// TwinCAT 3 PLC project BAUK_EK_BMS_PLC
// ProgramVersion: 3.1.4024.0
// libraries:
//   Recipe Management, * (System)
//   Tc2_BABasic, * (Beckhoff Automation GmbH)
//   Tc2_DALI, * (Beckhoff Automation GmbH)
//   Tc2_Database, * (Beckhoff Automation GmbH)
//   Tc2_DMX, * (Beckhoff Automation GmbH)
//   Tc2_EnOcean, * (Beckhoff Automation GmbH)
//   Tc2_EtherCAT, * (Beckhoff Automation GmbH)
//   Tc2_SerialCom, * (Beckhoff Automation GmbH)
//   Tc2_Standard, * (Beckhoff Automation GmbH)
//   Tc2_System, * (Beckhoff Automation GmbH)
//   Tc2_Utilities, * (Beckhoff Automation GmbH)
//   Tc3_DALI, * (Beckhoff Automation GmbH)
//   Tc3_IotBase, * (Beckhoff Automation GmbH)
//   Tc3_JsonXml, * (Beckhoff Automation GmbH)
//   Tc3_MLL, * (Beckhoff Automation GmbH)
//   Tc3_Module, * (Beckhoff Automation GmbH)
// project tree:
//   BLINDS/ ADSReadCX9020.TcPOU, BackgroundComms.TcPOU, BlindControl.TcPOU (not stored), BlindStretch.TcPOU, ConvertBoolArrayToString.TcPOU, fConvertBoolArrayToString.TcPOU, PrgMqttCom_Blinds_Publisher.TcPOU, Selection.TcDUT (not stored), StructAdvancedBlindControl.TcDUT (not stored), StructBlindControl.TcDUT (not stored)
//   ENOCEAN/ EnOcean.TcPOU
//   / FastDmxUpdate.TcTTO, Global_Variables.TcGVL, MAIN.TcPOU, PlcTask.TcTTO (not stored)
//   HMI/ FileHandle.TcPOU, ReadCP67.TcPOU, ST_SignInTable.TcDUT (not stored), SwitchTable.TcDUT (not stored), TableTennisScoreCounter.TcPOU, TIMESTR_Strings.TcDUT, VariableHandleForHmi.TcPOU
//   LIGHTS/DALI/ Dali.TcPOU, LightControl.TcPOU, LightTable.TcDUT (not stored)
//   LIGHTS/DMX/ DMX.TcPOU, ST_RGB.TcDUT
//   ML/ CoffeePredictionML.TcPOU (not stored), FB_CoffeeFifo.TcPOU, MLtest.TcPOU (not stored)
//   POWER MONITORING/ CoffeType.TcDUT (not stored), FB_Latch.TcPOU (not stored), PrgMqttCom_PM_Subscriber.TcPOU, SQLDB.TcPOU (not stored), ST_EL3403_Data.TcDUT, ST_PHASE_DATA.TcDUT (not stored)
//   WIND TURBINE/ FB_SendWhatsappCallMeBot.TcPOU, FB_WeatherAPI_HTTP.TcPOU, FB_WatsAppResponse.TcPOU, FB_WindTurbineSim.TcPOU
//   WORKSHOP WALL/ PowerSupply.TcPOU, Pulse.TcPOU, ST_PsuDiagData.TcDUT, ST_PsuInfoData.TcDUT
// real-time tasks:
//   TASK PlcTask: cycle T#2ms, priority 20, ADS port 350
//   TASK FastDmxUpdate: cycle T#1ms, priority 1, ADS port 351
// I/O:
//   DEVICE CX2040 E-Bus, AmsNetId 192.168.56.1.2.1
//     CX2040 Supply [EK1200-5000 EtherCAT Power supply (2A E-Bus)]
//       Server Room EtherCAT Junction [EK1122 2 port EtherCAT junction]
//         Boardroom DMX Node [EK1100 EtherCAT Coupler (2A E-Bus)]
//           Cabinet LED Strip Control [EL6851 DMX Master]
//           Term 17 (EL9011) [EL9011 End Terminal]
//         24Vdc Power Supply On Test Wall [PS2001-2410-1001 Power supply (24V, 10A, 1-phase)]
//         OLD BLIND CONTROL [EK1100 EtherCAT Coupler (2A E-Bus)] (disabled)
//           Coffee Machine Power Monitor [EL3403 3Ch. Power Measuring]
//           Blind Control Staff Room [EL6001 Interface (RS232)]
//           Blind Control Communal Area [EL6001 Interface (RS232)]
//           Blind Control Boardroom [EL6001 Interface (RS232)]
//       E-Bus to K-Bus
// variable links:
//   BAUK_EK_BMS_PLC/BAUK_EK_BMS_PLC Instance <-> CX2040 E-Bus/CX2040 Supply/E-Bus to K-Bus
//     PlcTask Inputs/.stDALIInData/nData <-> Office DALI Light Control/Channel 1/Data In
//     PlcTask Inputs/.stDALIInData/nStatus <-> Office DALI Light Control/Channel 1/State
//     PlcTask Inputs/.stKL6581InData/CNODE <-> Office EnOcean Switch Control/Channel 1/Input CNODE
//     PlcTask Inputs/.stKL6581InData/DB{0..3} <-> Office EnOcean Switch Control/Channel 1/Input DB{0..3}  (4 links)
//     PlcTask Inputs/.stKL6581InData/ID{0..3} <-> Office EnOcean Switch Control/Channel 1/Input ID{0..3}  (4 links)
//     PlcTask Inputs/.stKL6581InData/ORG <-> Office EnOcean Switch Control/Channel 1/Input ORG
//     PlcTask Inputs/.stKL6581InData/STATUS <-> Office EnOcean Switch Control/Channel 1/Input STATUS
//     PlcTask Inputs/.stKL6581InData/nStatus <-> Office EnOcean Switch Control/Channel 1/Status
//     PlcTask Inputs/.stKL6811InData/nData <-> Office DALI Light Control/Channel 1/Data In
//     PlcTask Inputs/.stKL6811InData/nStatus <-> Office DALI Light Control/Channel 1/State
//     PlcTask Inputs/EnOcean.STEnOceanInData/nData <-> Office RS485 EnOcean Control/Channel 1/Data In 0
//     PlcTask Inputs/EnOcean.STEnOceanInData/nData @bit {8..80 step 8} <-> Office RS485 EnOcean Control/Channel 1/Data In {1..10}  (10 links)
//     PlcTask Inputs/EnOcean.STEnOceanInData/nStatus <-> Office RS485 EnOcean Control/Channel 1/Ser. State
//     PlcTask Outputs/.stDALIOutData/nCtrl <-> Office DALI Light Control/Channel 1/Ctrl
//     PlcTask Outputs/.stDALIOutData/nData <-> Office DALI Light Control/Channel 1/Data Out
//     PlcTask Outputs/.stKL6581OutData/CNODE <-> Office EnOcean Switch Control/Channel 1/Output CNODE
//     PlcTask Outputs/.stKL6581OutData/DB{0..3} <-> Office EnOcean Switch Control/Channel 1/Output DB{0..3}  (4 links)
//     PlcTask Outputs/.stKL6581OutData/ID{0..3} <-> Office EnOcean Switch Control/Channel 1/Output ID{0..3}  (4 links)
//     PlcTask Outputs/.stKL6581OutData/ORG <-> Office EnOcean Switch Control/Channel 1/Output ORG
//     PlcTask Outputs/.stKL6581OutData/STATUS <-> Office EnOcean Switch Control/Channel 1/Output STATUS
//     PlcTask Outputs/.stKL6581OutData/nControl <-> Office EnOcean Switch Control/Channel 1/Control
//     PlcTask Outputs/EnOcean.STEnOceanOutData/nCtrl <-> Office RS485 EnOcean Control/Channel 1/Ser. Ctrl
//     PlcTask Outputs/EnOcean.STEnOceanOutData/nData[{0..10}] <-> Office RS485 EnOcean Control/Channel 1/Data Out {0..10}  (11 links)
//   BAUK_EK_BMS_PLC/BAUK_EK_BMS_PLC Instance <-> CX2040 E-Bus/CX2040 Supply/Server Room EtherCAT Junction/24Vdc Power Supply On Test Wall
//     PlcTask Inputs/PowerSupply.amsAdr <-> InfoData/AdsAddr
//     PlcTask Inputs/PowerSupply.psuDcOk <-> PSU Inputs/DC OK
//     PlcTask Inputs/PowerSupply.psuError <-> PSU Inputs/Error
//     PlcTask Inputs/PowerSupply.psuInputUnderVoltage <-> PSU Inputs Device/Input undervoltage
//     PlcTask Inputs/PowerSupply.psuOutCurrent <-> PSU Inputs/Output current
//     PlcTask Inputs/PowerSupply.psuOutVoltage <-> PSU Inputs/Output voltage
//     PlcTask Inputs/PowerSupply.psuWarning <-> PSU Inputs/Warning
//     PlcTask Outputs/PowerSupply.psuDisableOutput <-> PSU Outputs/Disable output
//   BAUK_EK_BMS_PLC/BAUK_EK_BMS_PLC Instance <-> CX2040 E-Bus/CX2040 Supply/Server Room EtherCAT Junction/Boardroom DMX Node/Cabinet LED Strip Control
//     FastDmxUpdate Inputs/.stDMXInDataLinie01/bCyclicTxDDisabled <-> DMX Status/Cyclic TxD disabled
//     FastDmxUpdate Inputs/.stDMXInDataLinie01/bDefaultDataSent <-> DMX Status/Default data sent
//     FastDmxUpdate Inputs/.stDMXInDataLinie01/bFrameSentToggle <-> DMX Status/Frame sent toggle
//     FastDmxUpdate Inputs/.stDMXInDataLinie01/bReceiveToggle <-> DMX Status/Receive toggle
//     FastDmxUpdate Inputs/.stDMXInDataLinie01/bTransmitAccepted <-> DMX Status/Transmit accepted
//     FastDmxUpdate Inputs/.stDMXInDataLinie01/bTxPDOToggle <-> DMX Status/TxPDO Toggle
//     FastDmxUpdate Inputs/.stDMXInDataLinie01/byStartCode <-> DMX Status/Start code
//     FastDmxUpdate Inputs/.stDMXInDataLinie01/wChannelLength <-> DMX Status/Channel length
//     FastDmxUpdate Outputs/.stDMXOutDataLinie01/arrData <-> DMX Channel 1-64/Channel 1
//     FastDmxUpdate Outputs/.stDMXOutDataLinie01/arrData @bit 72 <-> DMX Channel 1-64/Channel 10
//     FastDmxUpdate Outputs/.stDMXOutDataLinie01/arrData @bit 80 <-> DMX Channel 1-64/Channel 11
//     FastDmxUpdate Outputs/.stDMXOutDataLinie01/arrData @bit 88 <-> DMX Channel 1-64/Channel 12
//     FastDmxUpdate Outputs/.stDMXOutDataLinie01/arrData @bit 96 <-> DMX Channel 1-64/Channel 13
//     FastDmxUpdate Outputs/.stDMXOutDataLinie01/arrData @bit 104 <-> DMX Channel 1-64/Channel 14
//     FastDmxUpdate Outputs/.stDMXOutDataLinie01/arrData @bit 112 <-> DMX Channel 1-64/Channel 15
//     FastDmxUpdate Outputs/.stDMXOutDataLinie01/arrData @bit 120 <-> DMX Channel 1-64/Channel 16
//     FastDmxUpdate Outputs/.stDMXOutDataLinie01/arrData @bit 128 <-> DMX Channel 1-64/Channel 17
//     FastDmxUpdate Outputs/.stDMXOutDataLinie01/arrData @bit 136 <-> DMX Channel 1-64/Channel 18
//     FastDmxUpdate Outputs/.stDMXOutDataLinie01/arrData @bit 144 <-> DMX Channel 1-64/Channel 19
//     FastDmxUpdate Outputs/.stDMXOutDataLinie01/arrData @bit 8 <-> DMX Channel 1-64/Channel 2
//     FastDmxUpdate Outputs/.stDMXOutDataLinie01/arrData @bit 152 <-> DMX Channel 1-64/Channel 20
//     FastDmxUpdate Outputs/.stDMXOutDataLinie01/arrData @bit 160 <-> DMX Channel 1-64/Channel 21
//     FastDmxUpdate Outputs/.stDMXOutDataLinie01/arrData @bit 168 <-> DMX Channel 1-64/Channel 22
//     FastDmxUpdate Outputs/.stDMXOutDataLinie01/arrData @bit 176 <-> DMX Channel 1-64/Channel 23
//     FastDmxUpdate Outputs/.stDMXOutDataLinie01/arrData @bit 184 <-> DMX Channel 1-64/Channel 24
//     FastDmxUpdate Outputs/.stDMXOutDataLinie01/arrData @bit 192 <-> DMX Channel 1-64/Channel 25
//     FastDmxUpdate Outputs/.stDMXOutDataLinie01/arrData @bit 200 <-> DMX Channel 1-64/Channel 26
//     FastDmxUpdate Outputs/.stDMXOutDataLinie01/arrData @bit 208 <-> DMX Channel 1-64/Channel 27
//     FastDmxUpdate Outputs/.stDMXOutDataLinie01/arrData @bit 216 <-> DMX Channel 1-64/Channel 28
//     FastDmxUpdate Outputs/.stDMXOutDataLinie01/arrData @bit 224 <-> DMX Channel 1-64/Channel 29
//     FastDmxUpdate Outputs/.stDMXOutDataLinie01/arrData @bit 16 <-> DMX Channel 1-64/Channel 3
//     FastDmxUpdate Outputs/.stDMXOutDataLinie01/arrData @bit 232 <-> DMX Channel 1-64/Channel 30
//     FastDmxUpdate Outputs/.stDMXOutDataLinie01/arrData @bit 240 <-> DMX Channel 1-64/Channel 31
//     FastDmxUpdate Outputs/.stDMXOutDataLinie01/arrData @bit 248 <-> DMX Channel 1-64/Channel 32
//     FastDmxUpdate Outputs/.stDMXOutDataLinie01/arrData @bit 256 <-> DMX Channel 1-64/Channel 33
//     FastDmxUpdate Outputs/.stDMXOutDataLinie01/arrData @bit 264 <-> DMX Channel 1-64/Channel 34
//     FastDmxUpdate Outputs/.stDMXOutDataLinie01/arrData @bit 272 <-> DMX Channel 1-64/Channel 35
//     FastDmxUpdate Outputs/.stDMXOutDataLinie01/arrData @bit 280 <-> DMX Channel 1-64/Channel 36
//     FastDmxUpdate Outputs/.stDMXOutDataLinie01/arrData @bit 288 <-> DMX Channel 1-64/Channel 37
//     FastDmxUpdate Outputs/.stDMXOutDataLinie01/arrData @bit 296 <-> DMX Channel 1-64/Channel 38
//     FastDmxUpdate Outputs/.stDMXOutDataLinie01/arrData @bit 304 <-> DMX Channel 1-64/Channel 39
//     FastDmxUpdate Outputs/.stDMXOutDataLinie01/arrData @bit 24 <-> DMX Channel 1-64/Channel 4
//     FastDmxUpdate Outputs/.stDMXOutDataLinie01/arrData @bit 312 <-> DMX Channel 1-64/Channel 40
//     FastDmxUpdate Outputs/.stDMXOutDataLinie01/arrData @bit 320 <-> DMX Channel 1-64/Channel 41
//     FastDmxUpdate Outputs/.stDMXOutDataLinie01/arrData @bit 328 <-> DMX Channel 1-64/Channel 42
//     FastDmxUpdate Outputs/.stDMXOutDataLinie01/arrData @bit 336 <-> DMX Channel 1-64/Channel 43
//     FastDmxUpdate Outputs/.stDMXOutDataLinie01/arrData @bit 344 <-> DMX Channel 1-64/Channel 44
//     FastDmxUpdate Outputs/.stDMXOutDataLinie01/arrData @bit 352 <-> DMX Channel 1-64/Channel 45
//     FastDmxUpdate Outputs/.stDMXOutDataLinie01/arrData @bit 360 <-> DMX Channel 1-64/Channel 46
//     FastDmxUpdate Outputs/.stDMXOutDataLinie01/arrData @bit 368 <-> DMX Channel 1-64/Channel 47
//     FastDmxUpdate Outputs/.stDMXOutDataLinie01/arrData @bit 376 <-> DMX Channel 1-64/Channel 48
//     FastDmxUpdate Outputs/.stDMXOutDataLinie01/arrData @bit 384 <-> DMX Channel 1-64/Channel 49
//     FastDmxUpdate Outputs/.stDMXOutDataLinie01/arrData @bit 32 <-> DMX Channel 1-64/Channel 5
//     FastDmxUpdate Outputs/.stDMXOutDataLinie01/arrData @bit 392 <-> DMX Channel 1-64/Channel 50
//     FastDmxUpdate Outputs/.stDMXOutDataLinie01/arrData @bit 400 <-> DMX Channel 1-64/Channel 51
//     FastDmxUpdate Outputs/.stDMXOutDataLinie01/arrData @bit 408 <-> DMX Channel 1-64/Channel 52
//     FastDmxUpdate Outputs/.stDMXOutDataLinie01/arrData @bit 416 <-> DMX Channel 1-64/Channel 53
//     FastDmxUpdate Outputs/.stDMXOutDataLinie01/arrData @bit 424 <-> DMX Channel 1-64/Channel 54
//     FastDmxUpdate Outputs/.stDMXOutDataLinie01/arrData @bit 432 <-> DMX Channel 1-64/Channel 55
//     FastDmxUpdate Outputs/.stDMXOutDataLinie01/arrData @bit 440 <-> DMX Channel 1-64/Channel 56
//     FastDmxUpdate Outputs/.stDMXOutDataLinie01/arrData @bit 448 <-> DMX Channel 1-64/Channel 57
//     FastDmxUpdate Outputs/.stDMXOutDataLinie01/arrData @bit 456 <-> DMX Channel 1-64/Channel 58
//     FastDmxUpdate Outputs/.stDMXOutDataLinie01/arrData @bit 464 <-> DMX Channel 1-64/Channel 59
//     FastDmxUpdate Outputs/.stDMXOutDataLinie01/arrData @bit 40 <-> DMX Channel 1-64/Channel 6
//     FastDmxUpdate Outputs/.stDMXOutDataLinie01/arrData @bit 472 <-> DMX Channel 1-64/Channel 60
//     FastDmxUpdate Outputs/.stDMXOutDataLinie01/arrData @bit 480 <-> DMX Channel 1-64/Channel 61
//     FastDmxUpdate Outputs/.stDMXOutDataLinie01/arrData @bit 488 <-> DMX Channel 1-64/Channel 62
//     FastDmxUpdate Outputs/.stDMXOutDataLinie01/arrData @bit 496 <-> DMX Channel 1-64/Channel 63
//     FastDmxUpdate Outputs/.stDMXOutDataLinie01/arrData @bit 504 <-> DMX Channel 1-64/Channel 64
//     FastDmxUpdate Outputs/.stDMXOutDataLinie01/arrData @bit 48 <-> DMX Channel 1-64/Channel 7
//     FastDmxUpdate Outputs/.stDMXOutDataLinie01/arrData @bit 56 <-> DMX Channel 1-64/Channel 8
//     FastDmxUpdate Outputs/.stDMXOutDataLinie01/arrData @bit 64 <-> DMX Channel 1-64/Channel 9
//     FastDmxUpdate Outputs/.stDMXOutDataLinie01/arrData @bit 1024 <-> DMX Channel 129-192/Channel 129
//     FastDmxUpdate Outputs/.stDMXOutDataLinie01/arrData @bit 1032 <-> DMX Channel 129-192/Channel 130
//     FastDmxUpdate Outputs/.stDMXOutDataLinie01/arrData @bit 1040 <-> DMX Channel 129-192/Channel 131
//     FastDmxUpdate Outputs/.stDMXOutDataLinie01/arrData @bit 1048 <-> DMX Channel 129-192/Channel 132
//     FastDmxUpdate Outputs/.stDMXOutDataLinie01/arrData @bit 1056 <-> DMX Channel 129-192/Channel 133
//     FastDmxUpdate Outputs/.stDMXOutDataLinie01/arrData @bit 1064 <-> DMX Channel 129-192/Channel 134
//     FastDmxUpdate Outputs/.stDMXOutDataLinie01/arrData @bit 1072 <-> DMX Channel 129-192/Channel 135
//     FastDmxUpdate Outputs/.stDMXOutDataLinie01/arrData @bit 1080 <-> DMX Channel 129-192/Channel 136
//     FastDmxUpdate Outputs/.stDMXOutDataLinie01/arrData @bit 1088 <-> DMX Channel 129-192/Channel 137
//     FastDmxUpdate Outputs/.stDMXOutDataLinie01/arrData @bit 1096 <-> DMX Channel 129-192/Channel 138
//     FastDmxUpdate Outputs/.stDMXOutDataLinie01/arrData @bit 1104 <-> DMX Channel 129-192/Channel 139
//     FastDmxUpdate Outputs/.stDMXOutDataLinie01/arrData @bit 1112 <-> DMX Channel 129-192/Channel 140
//     FastDmxUpdate Outputs/.stDMXOutDataLinie01/arrData @bit 1120 <-> DMX Channel 129-192/Channel 141
//     FastDmxUpdate Outputs/.stDMXOutDataLinie01/arrData @bit 1128 <-> DMX Channel 129-192/Channel 142
//     FastDmxUpdate Outputs/.stDMXOutDataLinie01/arrData @bit 1136 <-> DMX Channel 129-192/Channel 143
//     FastDmxUpdate Outputs/.stDMXOutDataLinie01/arrData @bit 1144 <-> DMX Channel 129-192/Channel 144
//     FastDmxUpdate Outputs/.stDMXOutDataLinie01/arrData @bit 1152 <-> DMX Channel 129-192/Channel 145
//     FastDmxUpdate Outputs/.stDMXOutDataLinie01/arrData @bit 1160 <-> DMX Channel 129-192/Channel 146
//     FastDmxUpdate Outputs/.stDMXOutDataLinie01/arrData @bit 1168 <-> DMX Channel 129-192/Channel 147
//     FastDmxUpdate Outputs/.stDMXOutDataLinie01/arrData @bit 1176 <-> DMX Channel 129-192/Channel 148
//     FastDmxUpdate Outputs/.stDMXOutDataLinie01/arrData @bit 1184 <-> DMX Channel 129-192/Channel 149
//     FastDmxUpdate Outputs/.stDMXOutDataLinie01/arrData @bit 1192 <-> DMX Channel 129-192/Channel 150
//     FastDmxUpdate Outputs/.stDMXOutDataLinie01/arrData @bit 1200 <-> DMX Channel 129-192/Channel 151
//     FastDmxUpdate Outputs/.stDMXOutDataLinie01/arrData @bit 1208 <-> DMX Channel 129-192/Channel 152
//     FastDmxUpdate Outputs/.stDMXOutDataLinie01/arrData @bit 1216 <-> DMX Channel 129-192/Channel 153
//     FastDmxUpdate Outputs/.stDMXOutDataLinie01/arrData @bit 1224 <-> DMX Channel 129-192/Channel 154
//     FastDmxUpdate Outputs/.stDMXOutDataLinie01/arrData @bit 1232 <-> DMX Channel 129-192/Channel 155
//     FastDmxUpdate Outputs/.stDMXOutDataLinie01/arrData @bit 1240 <-> DMX Channel 129-192/Channel 156
//     FastDmxUpdate Outputs/.stDMXOutDataLinie01/arrData @bit 1248 <-> DMX Channel 129-192/Channel 157
//     FastDmxUpdate Outputs/.stDMXOutDataLinie01/arrData @bit 1256 <-> DMX Channel 129-192/Channel 158
//     FastDmxUpdate Outputs/.stDMXOutDataLinie01/arrData @bit 1264 <-> DMX Channel 129-192/Channel 159
//     FastDmxUpdate Outputs/.stDMXOutDataLinie01/arrData @bit 1272 <-> DMX Channel 129-192/Channel 160
//     FastDmxUpdate Outputs/.stDMXOutDataLinie01/arrData @bit 1280 <-> DMX Channel 129-192/Channel 161
//     FastDmxUpdate Outputs/.stDMXOutDataLinie01/arrData @bit 1288 <-> DMX Channel 129-192/Channel 162
//     FastDmxUpdate Outputs/.stDMXOutDataLinie01/arrData @bit 1296 <-> DMX Channel 129-192/Channel 163
//     FastDmxUpdate Outputs/.stDMXOutDataLinie01/arrData @bit 1304 <-> DMX Channel 129-192/Channel 164
//     FastDmxUpdate Outputs/.stDMXOutDataLinie01/arrData @bit 1312 <-> DMX Channel 129-192/Channel 165
//     FastDmxUpdate Outputs/.stDMXOutDataLinie01/arrData @bit 1320 <-> DMX Channel 129-192/Channel 166
//     FastDmxUpdate Outputs/.stDMXOutDataLinie01/arrData @bit 1328 <-> DMX Channel 129-192/Channel 167
//     FastDmxUpdate Outputs/.stDMXOutDataLinie01/arrData @bit 1336 <-> DMX Channel 129-192/Channel 168
//     FastDmxUpdate Outputs/.stDMXOutDataLinie01/arrData @bit 1344 <-> DMX Channel 129-192/Channel 169
//     FastDmxUpdate Outputs/.stDMXOutDataLinie01/arrData @bit 1352 <-> DMX Channel 129-192/Channel 170
//     FastDmxUpdate Outputs/.stDMXOutDataLinie01/arrData @bit 1360 <-> DMX Channel 129-192/Channel 171
//     FastDmxUpdate Outputs/.stDMXOutDataLinie01/arrData @bit 1368 <-> DMX Channel 129-192/Channel 172
//     FastDmxUpdate Outputs/.stDMXOutDataLinie01/arrData @bit 1376 <-> DMX Channel 129-192/Channel 173
//     FastDmxUpdate Outputs/.stDMXOutDataLinie01/arrData @bit 1384 <-> DMX Channel 129-192/Channel 174
//     FastDmxUpdate Outputs/.stDMXOutDataLinie01/arrData @bit 1392 <-> DMX Channel 129-192/Channel 175
//     FastDmxUpdate Outputs/.stDMXOutDataLinie01/arrData @bit 1400 <-> DMX Channel 129-192/Channel 176
//     FastDmxUpdate Outputs/.stDMXOutDataLinie01/arrData @bit 1408 <-> DMX Channel 129-192/Channel 177
//     FastDmxUpdate Outputs/.stDMXOutDataLinie01/arrData @bit 1416 <-> DMX Channel 129-192/Channel 178
//     FastDmxUpdate Outputs/.stDMXOutDataLinie01/arrData @bit 1424 <-> DMX Channel 129-192/Channel 179
//     FastDmxUpdate Outputs/.stDMXOutDataLinie01/arrData @bit 1432 <-> DMX Channel 129-192/Channel 180
//     FastDmxUpdate Outputs/.stDMXOutDataLinie01/arrData @bit 1440 <-> DMX Channel 129-192/Channel 181
//     FastDmxUpdate Outputs/.stDMXOutDataLinie01/arrData @bit 1448 <-> DMX Channel 129-192/Channel 182
//     FastDmxUpdate Outputs/.stDMXOutDataLinie01/arrData @bit 1456 <-> DMX Channel 129-192/Channel 183
//     FastDmxUpdate Outputs/.stDMXOutDataLinie01/arrData @bit 1464 <-> DMX Channel 129-192/Channel 184
//     FastDmxUpdate Outputs/.stDMXOutDataLinie01/arrData @bit 1472 <-> DMX Channel 129-192/Channel 185
//     FastDmxUpdate Outputs/.stDMXOutDataLinie01/arrData @bit 1480 <-> DMX Channel 129-192/Channel 186
//     FastDmxUpdate Outputs/.stDMXOutDataLinie01/arrData @bit 1488 <-> DMX Channel 129-192/Channel 187
//     FastDmxUpdate Outputs/.stDMXOutDataLinie01/arrData @bit 1496 <-> DMX Channel 129-192/Channel 188
//     FastDmxUpdate Outputs/.stDMXOutDataLinie01/arrData @bit 1504 <-> DMX Channel 129-192/Channel 189
//     FastDmxUpdate Outputs/.stDMXOutDataLinie01/arrData @bit 1512 <-> DMX Channel 129-192/Channel 190
//     FastDmxUpdate Outputs/.stDMXOutDataLinie01/arrData @bit 1520 <-> DMX Channel 129-192/Channel 191
//     FastDmxUpdate Outputs/.stDMXOutDataLinie01/arrData @bit 1528 <-> DMX Channel 129-192/Channel 192
//     FastDmxUpdate Outputs/.stDMXOutDataLinie01/arrData @bit 1536 <-> DMX Channel 193-256/Channel 193
//     FastDmxUpdate Outputs/.stDMXOutDataLinie01/arrData @bit 1544 <-> DMX Channel 193-256/Channel 194
//     FastDmxUpdate Outputs/.stDMXOutDataLinie01/arrData @bit 1552 <-> DMX Channel 193-256/Channel 195
//     FastDmxUpdate Outputs/.stDMXOutDataLinie01/arrData @bit 1560 <-> DMX Channel 193-256/Channel 196
//     FastDmxUpdate Outputs/.stDMXOutDataLinie01/arrData @bit 1568 <-> DMX Channel 193-256/Channel 197
//     FastDmxUpdate Outputs/.stDMXOutDataLinie01/arrData @bit 1576 <-> DMX Channel 193-256/Channel 198
//     FastDmxUpdate Outputs/.stDMXOutDataLinie01/arrData @bit 1584 <-> DMX Channel 193-256/Channel 199
//     FastDmxUpdate Outputs/.stDMXOutDataLinie01/arrData @bit 1592 <-> DMX Channel 193-256/Channel 200
//     FastDmxUpdate Outputs/.stDMXOutDataLinie01/arrData @bit 1600 <-> DMX Channel 193-256/Channel 201
//     FastDmxUpdate Outputs/.stDMXOutDataLinie01/arrData @bit 1608 <-> DMX Channel 193-256/Channel 202
//     FastDmxUpdate Outputs/.stDMXOutDataLinie01/arrData @bit 1616 <-> DMX Channel 193-256/Channel 203
//     FastDmxUpdate Outputs/.stDMXOutDataLinie01/arrData @bit 1624 <-> DMX Channel 193-256/Channel 204
//     FastDmxUpdate Outputs/.stDMXOutDataLinie01/arrData @bit 1632 <-> DMX Channel 193-256/Channel 205
//     FastDmxUpdate Outputs/.stDMXOutDataLinie01/arrData @bit 1640 <-> DMX Channel 193-256/Channel 206
//     FastDmxUpdate Outputs/.stDMXOutDataLinie01/arrData @bit 1648 <-> DMX Channel 193-256/Channel 207
//     FastDmxUpdate Outputs/.stDMXOutDataLinie01/arrData @bit 1656 <-> DMX Channel 193-256/Channel 208
//     FastDmxUpdate Outputs/.stDMXOutDataLinie01/arrData @bit 1664 <-> DMX Channel 193-256/Channel 209
//     FastDmxUpdate Outputs/.stDMXOutDataLinie01/arrData @bit 1672 <-> DMX Channel 193-256/Channel 210
//     FastDmxUpdate Outputs/.stDMXOutDataLinie01/arrData @bit 1680 <-> DMX Channel 193-256/Channel 211
//     FastDmxUpdate Outputs/.stDMXOutDataLinie01/arrData @bit 1688 <-> DMX Channel 193-256/Channel 212
//     FastDmxUpdate Outputs/.stDMXOutDataLinie01/arrData @bit 1696 <-> DMX Channel 193-256/Channel 213
//     FastDmxUpdate Outputs/.stDMXOutDataLinie01/arrData @bit 1704 <-> DMX Channel 193-256/Channel 214
//     FastDmxUpdate Outputs/.stDMXOutDataLinie01/arrData @bit 1712 <-> DMX Channel 193-256/Channel 215
//     FastDmxUpdate Outputs/.stDMXOutDataLinie01/arrData @bit 1720 <-> DMX Channel 193-256/Channel 216
//     FastDmxUpdate Outputs/.stDMXOutDataLinie01/arrData @bit 1728 <-> DMX Channel 193-256/Channel 217
//     FastDmxUpdate Outputs/.stDMXOutDataLinie01/arrData @bit 1736 <-> DMX Channel 193-256/Channel 218
//     FastDmxUpdate Outputs/.stDMXOutDataLinie01/arrData @bit 1744 <-> DMX Channel 193-256/Channel 219
//     FastDmxUpdate Outputs/.stDMXOutDataLinie01/arrData @bit 1752 <-> DMX Channel 193-256/Channel 220
//     FastDmxUpdate Outputs/.stDMXOutDataLinie01/arrData @bit 1760 <-> DMX Channel 193-256/Channel 221
//     FastDmxUpdate Outputs/.stDMXOutDataLinie01/arrData @bit 1768 <-> DMX Channel 193-256/Channel 222
//     FastDmxUpdate Outputs/.stDMXOutDataLinie01/arrData @bit 1776 <-> DMX Channel 193-256/Channel 223
//     FastDmxUpdate Outputs/.stDMXOutDataLinie01/arrData @bit 1784 <-> DMX Channel 193-256/Channel 224
//     FastDmxUpdate Outputs/.stDMXOutDataLinie01/arrData @bit 1792 <-> DMX Channel 193-256/Channel 225
//     FastDmxUpdate Outputs/.stDMXOutDataLinie01/arrData @bit 1800 <-> DMX Channel 193-256/Channel 226
//     FastDmxUpdate Outputs/.stDMXOutDataLinie01/arrData @bit 1808 <-> DMX Channel 193-256/Channel 227
//     FastDmxUpdate Outputs/.stDMXOutDataLinie01/arrData @bit 1816 <-> DMX Channel 193-256/Channel 228
//     FastDmxUpdate Outputs/.stDMXOutDataLinie01/arrData @bit 1824 <-> DMX Channel 193-256/Channel 229
//     FastDmxUpdate Outputs/.stDMXOutDataLinie01/arrData @bit 1832 <-> DMX Channel 193-256/Channel 230
//     FastDmxUpdate Outputs/.stDMXOutDataLinie01/arrData @bit 1840 <-> DMX Channel 193-256/Channel 231
//     FastDmxUpdate Outputs/.stDMXOutDataLinie01/arrData @bit 1848 <-> DMX Channel 193-256/Channel 232
//     FastDmxUpdate Outputs/.stDMXOutDataLinie01/arrData @bit 1856 <-> DMX Channel 193-256/Channel 233
//     FastDmxUpdate Outputs/.stDMXOutDataLinie01/arrData @bit 1864 <-> DMX Channel 193-256/Channel 234
//     FastDmxUpdate Outputs/.stDMXOutDataLinie01/arrData @bit 1872 <-> DMX Channel 193-256/Channel 235
//     FastDmxUpdate Outputs/.stDMXOutDataLinie01/arrData @bit 1880 <-> DMX Channel 193-256/Channel 236
//     FastDmxUpdate Outputs/.stDMXOutDataLinie01/arrData @bit 1888 <-> DMX Channel 193-256/Channel 237
//     FastDmxUpdate Outputs/.stDMXOutDataLinie01/arrData @bit 1896 <-> DMX Channel 193-256/Channel 238
//     FastDmxUpdate Outputs/.stDMXOutDataLinie01/arrData @bit 1904 <-> DMX Channel 193-256/Channel 239
//     FastDmxUpdate Outputs/.stDMXOutDataLinie01/arrData @bit 1912 <-> DMX Channel 193-256/Channel 240
//     FastDmxUpdate Outputs/.stDMXOutDataLinie01/arrData @bit 1920 <-> DMX Channel 193-256/Channel 241
//     FastDmxUpdate Outputs/.stDMXOutDataLinie01/arrData @bit 1928 <-> DMX Channel 193-256/Channel 242
//     FastDmxUpdate Outputs/.stDMXOutDataLinie01/arrData @bit 1936 <-> DMX Channel 193-256/Channel 243
//     FastDmxUpdate Outputs/.stDMXOutDataLinie01/arrData @bit 1944 <-> DMX Channel 193-256/Channel 244
//     FastDmxUpdate Outputs/.stDMXOutDataLinie01/arrData @bit 1952 <-> DMX Channel 193-256/Channel 245
//     FastDmxUpdate Outputs/.stDMXOutDataLinie01/arrData @bit 1960 <-> DMX Channel 193-256/Channel 246
//     FastDmxUpdate Outputs/.stDMXOutDataLinie01/arrData @bit 1968 <-> DMX Channel 193-256/Channel 247
//     FastDmxUpdate Outputs/.stDMXOutDataLinie01/arrData @bit 1976 <-> DMX Channel 193-256/Channel 248
//     FastDmxUpdate Outputs/.stDMXOutDataLinie01/arrData @bit 1984 <-> DMX Channel 193-256/Channel 249
//     FastDmxUpdate Outputs/.stDMXOutDataLinie01/arrData @bit 1992 <-> DMX Channel 193-256/Channel 250
//     FastDmxUpdate Outputs/.stDMXOutDataLinie01/arrData @bit 2000 <-> DMX Channel 193-256/Channel 251
//     FastDmxUpdate Outputs/.stDMXOutDataLinie01/arrData @bit 2008 <-> DMX Channel 193-256/Channel 252
//     FastDmxUpdate Outputs/.stDMXOutDataLinie01/arrData @bit 2016 <-> DMX Channel 193-256/Channel 253
//     FastDmxUpdate Outputs/.stDMXOutDataLinie01/arrData @bit 2024 <-> DMX Channel 193-256/Channel 254
//     FastDmxUpdate Outputs/.stDMXOutDataLinie01/arrData @bit 2032 <-> DMX Channel 193-256/Channel 255
//     FastDmxUpdate Outputs/.stDMXOutDataLinie01/arrData @bit 2040 <-> DMX Channel 193-256/Channel 256
//     FastDmxUpdate Outputs/.stDMXOutDataLinie01/arrData @bit 2048 <-> DMX Channel 257-320/Channel 257
//     FastDmxUpdate Outputs/.stDMXOutDataLinie01/arrData @bit 2056 <-> DMX Channel 257-320/Channel 258
//     FastDmxUpdate Outputs/.stDMXOutDataLinie01/arrData @bit 2064 <-> DMX Channel 257-320/Channel 259
//     FastDmxUpdate Outputs/.stDMXOutDataLinie01/arrData @bit 2072 <-> DMX Channel 257-320/Channel 260
//     FastDmxUpdate Outputs/.stDMXOutDataLinie01/arrData @bit 2080 <-> DMX Channel 257-320/Channel 261
//     FastDmxUpdate Outputs/.stDMXOutDataLinie01/arrData @bit 2088 <-> DMX Channel 257-320/Channel 262
//     FastDmxUpdate Outputs/.stDMXOutDataLinie01/arrData @bit 2096 <-> DMX Channel 257-320/Channel 263
//     FastDmxUpdate Outputs/.stDMXOutDataLinie01/arrData @bit 2104 <-> DMX Channel 257-320/Channel 264
//     FastDmxUpdate Outputs/.stDMXOutDataLinie01/arrData @bit 2112 <-> DMX Channel 257-320/Channel 265
//     FastDmxUpdate Outputs/.stDMXOutDataLinie01/arrData @bit 2120 <-> DMX Channel 257-320/Channel 266
//     FastDmxUpdate Outputs/.stDMXOutDataLinie01/arrData @bit 2128 <-> DMX Channel 257-320/Channel 267
//     FastDmxUpdate Outputs/.stDMXOutDataLinie01/arrData @bit 2136 <-> DMX Channel 257-320/Channel 268
//     FastDmxUpdate Outputs/.stDMXOutDataLinie01/arrData @bit 2144 <-> DMX Channel 257-320/Channel 269
//     FastDmxUpdate Outputs/.stDMXOutDataLinie01/arrData @bit 2152 <-> DMX Channel 257-320/Channel 270
//     FastDmxUpdate Outputs/.stDMXOutDataLinie01/arrData @bit 2160 <-> DMX Channel 257-320/Channel 271
//     FastDmxUpdate Outputs/.stDMXOutDataLinie01/arrData @bit 2168 <-> DMX Channel 257-320/Channel 272
//     FastDmxUpdate Outputs/.stDMXOutDataLinie01/arrData @bit 2176 <-> DMX Channel 257-320/Channel 273
//     FastDmxUpdate Outputs/.stDMXOutDataLinie01/arrData @bit 2184 <-> DMX Channel 257-320/Channel 274
//     FastDmxUpdate Outputs/.stDMXOutDataLinie01/arrData @bit 2192 <-> DMX Channel 257-320/Channel 275
//     FastDmxUpdate Outputs/.stDMXOutDataLinie01/arrData @bit 2200 <-> DMX Channel 257-320/Channel 276
//     FastDmxUpdate Outputs/.stDMXOutDataLinie01/arrData @bit 2208 <-> DMX Channel 257-320/Channel 277
//     FastDmxUpdate Outputs/.stDMXOutDataLinie01/arrData @bit 2216 <-> DMX Channel 257-320/Channel 278
//     FastDmxUpdate Outputs/.stDMXOutDataLinie01/arrData @bit 2224 <-> DMX Channel 257-320/Channel 279
//     FastDmxUpdate Outputs/.stDMXOutDataLinie01/arrData @bit 2232 <-> DMX Channel 257-320/Channel 280
//     FastDmxUpdate Outputs/.stDMXOutDataLinie01/arrData @bit 2240 <-> DMX Channel 257-320/Channel 281
//     FastDmxUpdate Outputs/.stDMXOutDataLinie01/arrData @bit 2248 <-> DMX Channel 257-320/Channel 282
//     FastDmxUpdate Outputs/.stDMXOutDataLinie01/arrData @bit 2256 <-> DMX Channel 257-320/Channel 283
//     FastDmxUpdate Outputs/.stDMXOutDataLinie01/arrData @bit 2264 <-> DMX Channel 257-320/Channel 284
//     FastDmxUpdate Outputs/.stDMXOutDataLinie01/arrData @bit 2272 <-> DMX Channel 257-320/Channel 285
//     FastDmxUpdate Outputs/.stDMXOutDataLinie01/arrData @bit 2280 <-> DMX Channel 257-320/Channel 286
//     FastDmxUpdate Outputs/.stDMXOutDataLinie01/arrData @bit 2288 <-> DMX Channel 257-320/Channel 287
//     FastDmxUpdate Outputs/.stDMXOutDataLinie01/arrData @bit 2296 <-> DMX Channel 257-320/Channel 288
//     FastDmxUpdate Outputs/.stDMXOutDataLinie01/arrData @bit 2304 <-> DMX Channel 257-320/Channel 289
//     FastDmxUpdate Outputs/.stDMXOutDataLinie01/arrData @bit 2312 <-> DMX Channel 257-320/Channel 290
//     FastDmxUpdate Outputs/.stDMXOutDataLinie01/arrData @bit 2320 <-> DMX Channel 257-320/Channel 291
//     FastDmxUpdate Outputs/.stDMXOutDataLinie01/arrData @bit 2328 <-> DMX Channel 257-320/Channel 292
//     FastDmxUpdate Outputs/.stDMXOutDataLinie01/arrData @bit 2336 <-> DMX Channel 257-320/Channel 293
//     FastDmxUpdate Outputs/.stDMXOutDataLinie01/arrData @bit 2344 <-> DMX Channel 257-320/Channel 294
//     FastDmxUpdate Outputs/.stDMXOutDataLinie01/arrData @bit 2352 <-> DMX Channel 257-320/Channel 295
//     FastDmxUpdate Outputs/.stDMXOutDataLinie01/arrData @bit 2360 <-> DMX Channel 257-320/Channel 296
//     FastDmxUpdate Outputs/.stDMXOutDataLinie01/arrData @bit 2368 <-> DMX Channel 257-320/Channel 297
//     FastDmxUpdate Outputs/.stDMXOutDataLinie01/arrData @bit 2376 <-> DMX Channel 257-320/Channel 298
//     FastDmxUpdate Outputs/.stDMXOutDataLinie01/arrData @bit 2384 <-> DMX Channel 257-320/Channel 299
//     FastDmxUpdate Outputs/.stDMXOutDataLinie01/arrData @bit 2392 <-> DMX Channel 257-320/Channel 300
//     FastDmxUpdate Outputs/.stDMXOutDataLinie01/arrData @bit 2400 <-> DMX Channel 257-320/Channel 301
//     FastDmxUpdate Outputs/.stDMXOutDataLinie01/arrData @bit 2408 <-> DMX Channel 257-320/Channel 302
//     FastDmxUpdate Outputs/.stDMXOutDataLinie01/arrData @bit 2416 <-> DMX Channel 257-320/Channel 303
//     FastDmxUpdate Outputs/.stDMXOutDataLinie01/arrData @bit 2424 <-> DMX Channel 257-320/Channel 304
//     FastDmxUpdate Outputs/.stDMXOutDataLinie01/arrData @bit 2432 <-> DMX Channel 257-320/Channel 305
//     FastDmxUpdate Outputs/.stDMXOutDataLinie01/arrData @bit 2440 <-> DMX Channel 257-320/Channel 306
//     FastDmxUpdate Outputs/.stDMXOutDataLinie01/arrData @bit 2448 <-> DMX Channel 257-320/Channel 307
//     FastDmxUpdate Outputs/.stDMXOutDataLinie01/arrData @bit 2456 <-> DMX Channel 257-320/Channel 308
//     FastDmxUpdate Outputs/.stDMXOutDataLinie01/arrData @bit 2464 <-> DMX Channel 257-320/Channel 309
//     FastDmxUpdate Outputs/.stDMXOutDataLinie01/arrData @bit 2472 <-> DMX Channel 257-320/Channel 310
//     FastDmxUpdate Outputs/.stDMXOutDataLinie01/arrData @bit 2480 <-> DMX Channel 257-320/Channel 311
//     FastDmxUpdate Outputs/.stDMXOutDataLinie01/arrData @bit 2488 <-> DMX Channel 257-320/Channel 312
//     FastDmxUpdate Outputs/.stDMXOutDataLinie01/arrData @bit 2496 <-> DMX Channel 257-320/Channel 313
//     FastDmxUpdate Outputs/.stDMXOutDataLinie01/arrData @bit 2504 <-> DMX Channel 257-320/Channel 314
//     FastDmxUpdate Outputs/.stDMXOutDataLinie01/arrData @bit 2512 <-> DMX Channel 257-320/Channel 315
//     FastDmxUpdate Outputs/.stDMXOutDataLinie01/arrData @bit 2520 <-> DMX Channel 257-320/Channel 316
//     FastDmxUpdate Outputs/.stDMXOutDataLinie01/arrData @bit 2528 <-> DMX Channel 257-320/Channel 317
//     FastDmxUpdate Outputs/.stDMXOutDataLinie01/arrData @bit 2536 <-> DMX Channel 257-320/Channel 318
//     FastDmxUpdate Outputs/.stDMXOutDataLinie01/arrData @bit 2544 <-> DMX Channel 257-320/Channel 319
//     FastDmxUpdate Outputs/.stDMXOutDataLinie01/arrData @bit 2552 <-> DMX Channel 257-320/Channel 320
//     FastDmxUpdate Outputs/.stDMXOutDataLinie01/arrData @bit 2560 <-> DMX Channel 321-384/Channel 321
//     FastDmxUpdate Outputs/.stDMXOutDataLinie01/arrData @bit 2568 <-> DMX Channel 321-384/Channel 322
//     FastDmxUpdate Outputs/.stDMXOutDataLinie01/arrData @bit 2576 <-> DMX Channel 321-384/Channel 323
//     FastDmxUpdate Outputs/.stDMXOutDataLinie01/arrData @bit 2584 <-> DMX Channel 321-384/Channel 324
//     FastDmxUpdate Outputs/.stDMXOutDataLinie01/arrData @bit 2592 <-> DMX Channel 321-384/Channel 325
//     FastDmxUpdate Outputs/.stDMXOutDataLinie01/arrData @bit 2600 <-> DMX Channel 321-384/Channel 326
//     FastDmxUpdate Outputs/.stDMXOutDataLinie01/arrData @bit 2608 <-> DMX Channel 321-384/Channel 327
//     FastDmxUpdate Outputs/.stDMXOutDataLinie01/arrData @bit 2616 <-> DMX Channel 321-384/Channel 328
//     FastDmxUpdate Outputs/.stDMXOutDataLinie01/arrData @bit 2624 <-> DMX Channel 321-384/Channel 329
//     FastDmxUpdate Outputs/.stDMXOutDataLinie01/arrData @bit 2632 <-> DMX Channel 321-384/Channel 330
//     FastDmxUpdate Outputs/.stDMXOutDataLinie01/arrData @bit 2640 <-> DMX Channel 321-384/Channel 331
//     FastDmxUpdate Outputs/.stDMXOutDataLinie01/arrData @bit 2648 <-> DMX Channel 321-384/Channel 332
//     FastDmxUpdate Outputs/.stDMXOutDataLinie01/arrData @bit 2656 <-> DMX Channel 321-384/Channel 333
//     FastDmxUpdate Outputs/.stDMXOutDataLinie01/arrData @bit 2664 <-> DMX Channel 321-384/Channel 334
//     FastDmxUpdate Outputs/.stDMXOutDataLinie01/arrData @bit 2672 <-> DMX Channel 321-384/Channel 335
//     FastDmxUpdate Outputs/.stDMXOutDataLinie01/arrData @bit 2680 <-> DMX Channel 321-384/Channel 336
//     FastDmxUpdate Outputs/.stDMXOutDataLinie01/arrData @bit 2688 <-> DMX Channel 321-384/Channel 337
//     FastDmxUpdate Outputs/.stDMXOutDataLinie01/arrData @bit 2696 <-> DMX Channel 321-384/Channel 338
//     FastDmxUpdate Outputs/.stDMXOutDataLinie01/arrData @bit 2704 <-> DMX Channel 321-384/Channel 339
//     FastDmxUpdate Outputs/.stDMXOutDataLinie01/arrData @bit 2712 <-> DMX Channel 321-384/Channel 340
//     FastDmxUpdate Outputs/.stDMXOutDataLinie01/arrData @bit 2720 <-> DMX Channel 321-384/Channel 341
//     FastDmxUpdate Outputs/.stDMXOutDataLinie01/arrData @bit 2728 <-> DMX Channel 321-384/Channel 342
//     FastDmxUpdate Outputs/.stDMXOutDataLinie01/arrData @bit 2736 <-> DMX Channel 321-384/Channel 343
//     FastDmxUpdate Outputs/.stDMXOutDataLinie01/arrData @bit 2744 <-> DMX Channel 321-384/Channel 344
//     FastDmxUpdate Outputs/.stDMXOutDataLinie01/arrData @bit 2752 <-> DMX Channel 321-384/Channel 345
//     FastDmxUpdate Outputs/.stDMXOutDataLinie01/arrData @bit 2760 <-> DMX Channel 321-384/Channel 346
//     FastDmxUpdate Outputs/.stDMXOutDataLinie01/arrData @bit 2768 <-> DMX Channel 321-384/Channel 347
//     FastDmxUpdate Outputs/.stDMXOutDataLinie01/arrData @bit 2776 <-> DMX Channel 321-384/Channel 348
//     FastDmxUpdate Outputs/.stDMXOutDataLinie01/arrData @bit 2784 <-> DMX Channel 321-384/Channel 349
//     FastDmxUpdate Outputs/.stDMXOutDataLinie01/arrData @bit 2792 <-> DMX Channel 321-384/Channel 350
//     FastDmxUpdate Outputs/.stDMXOutDataLinie01/arrData @bit 2800 <-> DMX Channel 321-384/Channel 351
//     FastDmxUpdate Outputs/.stDMXOutDataLinie01/arrData @bit 2808 <-> DMX Channel 321-384/Channel 352
//     FastDmxUpdate Outputs/.stDMXOutDataLinie01/arrData @bit 2816 <-> DMX Channel 321-384/Channel 353
//     FastDmxUpdate Outputs/.stDMXOutDataLinie01/arrData @bit 2824 <-> DMX Channel 321-384/Channel 354
//     FastDmxUpdate Outputs/.stDMXOutDataLinie01/arrData @bit 2832 <-> DMX Channel 321-384/Channel 355
//     FastDmxUpdate Outputs/.stDMXOutDataLinie01/arrData @bit 2840 <-> DMX Channel 321-384/Channel 356
//     FastDmxUpdate Outputs/.stDMXOutDataLinie01/arrData @bit 2848 <-> DMX Channel 321-384/Channel 357
//     FastDmxUpdate Outputs/.stDMXOutDataLinie01/arrData @bit 2856 <-> DMX Channel 321-384/Channel 358
//     FastDmxUpdate Outputs/.stDMXOutDataLinie01/arrData @bit 2864 <-> DMX Channel 321-384/Channel 359
//     FastDmxUpdate Outputs/.stDMXOutDataLinie01/arrData @bit 2872 <-> DMX Channel 321-384/Channel 360
//     FastDmxUpdate Outputs/.stDMXOutDataLinie01/arrData @bit 2880 <-> DMX Channel 321-384/Channel 361
//     FastDmxUpdate Outputs/.stDMXOutDataLinie01/arrData @bit 2888 <-> DMX Channel 321-384/Channel 362
//     FastDmxUpdate Outputs/.stDMXOutDataLinie01/arrData @bit 2896 <-> DMX Channel 321-384/Channel 363
//     FastDmxUpdate Outputs/.stDMXOutDataLinie01/arrData @bit 2904 <-> DMX Channel 321-384/Channel 364
//     FastDmxUpdate Outputs/.stDMXOutDataLinie01/arrData @bit 2912 <-> DMX Channel 321-384/Channel 365
//     FastDmxUpdate Outputs/.stDMXOutDataLinie01/arrData @bit 2920 <-> DMX Channel 321-384/Channel 366
//     FastDmxUpdate Outputs/.stDMXOutDataLinie01/arrData @bit 2928 <-> DMX Channel 321-384/Channel 367
//     FastDmxUpdate Outputs/.stDMXOutDataLinie01/arrData @bit 2936 <-> DMX Channel 321-384/Channel 368
//     FastDmxUpdate Outputs/.stDMXOutDataLinie01/arrData @bit 2944 <-> DMX Channel 321-384/Channel 369
//     FastDmxUpdate Outputs/.stDMXOutDataLinie01/arrData @bit 2952 <-> DMX Channel 321-384/Channel 370
//     FastDmxUpdate Outputs/.stDMXOutDataLinie01/arrData @bit 2960 <-> DMX Channel 321-384/Channel 371
//     FastDmxUpdate Outputs/.stDMXOutDataLinie01/arrData @bit 2968 <-> DMX Channel 321-384/Channel 372
//     FastDmxUpdate Outputs/.stDMXOutDataLinie01/arrData @bit 2976 <-> DMX Channel 321-384/Channel 373
//     FastDmxUpdate Outputs/.stDMXOutDataLinie01/arrData @bit 2984 <-> DMX Channel 321-384/Channel 374
//     FastDmxUpdate Outputs/.stDMXOutDataLinie01/arrData @bit 2992 <-> DMX Channel 321-384/Channel 375
//     FastDmxUpdate Outputs/.stDMXOutDataLinie01/arrData @bit 3000 <-> DMX Channel 321-384/Channel 376
//     FastDmxUpdate Outputs/.stDMXOutDataLinie01/arrData @bit 3008 <-> DMX Channel 321-384/Channel 377
//     FastDmxUpdate Outputs/.stDMXOutDataLinie01/arrData @bit 3016 <-> DMX Channel 321-384/Channel 378
//     FastDmxUpdate Outputs/.stDMXOutDataLinie01/arrData @bit 3024 <-> DMX Channel 321-384/Channel 379
//     FastDmxUpdate Outputs/.stDMXOutDataLinie01/arrData @bit 3032 <-> DMX Channel 321-384/Channel 380
//     FastDmxUpdate Outputs/.stDMXOutDataLinie01/arrData @bit 3040 <-> DMX Channel 321-384/Channel 381
//     FastDmxUpdate Outputs/.stDMXOutDataLinie01/arrData @bit 3048 <-> DMX Channel 321-384/Channel 382
//     FastDmxUpdate Outputs/.stDMXOutDataLinie01/arrData @bit 3056 <-> DMX Channel 321-384/Channel 383
//     FastDmxUpdate Outputs/.stDMXOutDataLinie01/arrData @bit 3064 <-> DMX Channel 321-384/Channel 384
//     FastDmxUpdate Outputs/.stDMXOutDataLinie01/arrData @bit 3072 <-> DMX Channel 385-448/Channel 385
//     FastDmxUpdate Outputs/.stDMXOutDataLinie01/arrData @bit 3080 <-> DMX Channel 385-448/Channel 386
//     FastDmxUpdate Outputs/.stDMXOutDataLinie01/arrData @bit 3088 <-> DMX Channel 385-448/Channel 387
//     FastDmxUpdate Outputs/.stDMXOutDataLinie01/arrData @bit 3096 <-> DMX Channel 385-448/Channel 388
//     FastDmxUpdate Outputs/.stDMXOutDataLinie01/arrData @bit 3104 <-> DMX Channel 385-448/Channel 389
//     FastDmxUpdate Outputs/.stDMXOutDataLinie01/arrData @bit 3112 <-> DMX Channel 385-448/Channel 390
//     FastDmxUpdate Outputs/.stDMXOutDataLinie01/arrData @bit 3120 <-> DMX Channel 385-448/Channel 391
//     FastDmxUpdate Outputs/.stDMXOutDataLinie01/arrData @bit 3128 <-> DMX Channel 385-448/Channel 392
//     FastDmxUpdate Outputs/.stDMXOutDataLinie01/arrData @bit 3136 <-> DMX Channel 385-448/Channel 393
//     FastDmxUpdate Outputs/.stDMXOutDataLinie01/arrData @bit 3144 <-> DMX Channel 385-448/Channel 394
//     FastDmxUpdate Outputs/.stDMXOutDataLinie01/arrData @bit 3152 <-> DMX Channel 385-448/Channel 395
//     FastDmxUpdate Outputs/.stDMXOutDataLinie01/arrData @bit 3160 <-> DMX Channel 385-448/Channel 396
//     FastDmxUpdate Outputs/.stDMXOutDataLinie01/arrData @bit 3168 <-> DMX Channel 385-448/Channel 397
//     FastDmxUpdate Outputs/.stDMXOutDataLinie01/arrData @bit 3176 <-> DMX Channel 385-448/Channel 398
//     FastDmxUpdate Outputs/.stDMXOutDataLinie01/arrData @bit 3184 <-> DMX Channel 385-448/Channel 399
//     FastDmxUpdate Outputs/.stDMXOutDataLinie01/arrData @bit 3192 <-> DMX Channel 385-448/Channel 400
//     FastDmxUpdate Outputs/.stDMXOutDataLinie01/arrData @bit 3200 <-> DMX Channel 385-448/Channel 401
//     FastDmxUpdate Outputs/.stDMXOutDataLinie01/arrData @bit 3208 <-> DMX Channel 385-448/Channel 402
//     FastDmxUpdate Outputs/.stDMXOutDataLinie01/arrData @bit 3216 <-> DMX Channel 385-448/Channel 403
//     FastDmxUpdate Outputs/.stDMXOutDataLinie01/arrData @bit 3224 <-> DMX Channel 385-448/Channel 404
//     FastDmxUpdate Outputs/.stDMXOutDataLinie01/arrData @bit 3232 <-> DMX Channel 385-448/Channel 405
//     FastDmxUpdate Outputs/.stDMXOutDataLinie01/arrData @bit 3240 <-> DMX Channel 385-448/Channel 406
//     FastDmxUpdate Outputs/.stDMXOutDataLinie01/arrData @bit 3248 <-> DMX Channel 385-448/Channel 407
//     FastDmxUpdate Outputs/.stDMXOutDataLinie01/arrData @bit 3256 <-> DMX Channel 385-448/Channel 408
//     FastDmxUpdate Outputs/.stDMXOutDataLinie01/arrData @bit 3264 <-> DMX Channel 385-448/Channel 409
//     FastDmxUpdate Outputs/.stDMXOutDataLinie01/arrData @bit 3272 <-> DMX Channel 385-448/Channel 410
//     FastDmxUpdate Outputs/.stDMXOutDataLinie01/arrData @bit 3280 <-> DMX Channel 385-448/Channel 411
//     FastDmxUpdate Outputs/.stDMXOutDataLinie01/arrData @bit 3288 <-> DMX Channel 385-448/Channel 412
//     FastDmxUpdate Outputs/.stDMXOutDataLinie01/arrData @bit 3296 <-> DMX Channel 385-448/Channel 413
//     FastDmxUpdate Outputs/.stDMXOutDataLinie01/arrData @bit 3304 <-> DMX Channel 385-448/Channel 414
//     FastDmxUpdate Outputs/.stDMXOutDataLinie01/arrData @bit 3312 <-> DMX Channel 385-448/Channel 415
//     FastDmxUpdate Outputs/.stDMXOutDataLinie01/arrData @bit 3320 <-> DMX Channel 385-448/Channel 416
//     FastDmxUpdate Outputs/.stDMXOutDataLinie01/arrData @bit 3328 <-> DMX Channel 385-448/Channel 417
//     FastDmxUpdate Outputs/.stDMXOutDataLinie01/arrData @bit 3336 <-> DMX Channel 385-448/Channel 418
//     FastDmxUpdate Outputs/.stDMXOutDataLinie01/arrData @bit 3344 <-> DMX Channel 385-448/Channel 419
//     FastDmxUpdate Outputs/.stDMXOutDataLinie01/arrData @bit 3352 <-> DMX Channel 385-448/Channel 420
//     FastDmxUpdate Outputs/.stDMXOutDataLinie01/arrData @bit 3360 <-> DMX Channel 385-448/Channel 421
//     FastDmxUpdate Outputs/.stDMXOutDataLinie01/arrData @bit 3368 <-> DMX Channel 385-448/Channel 422
//     FastDmxUpdate Outputs/.stDMXOutDataLinie01/arrData @bit 3376 <-> DMX Channel 385-448/Channel 423
//     FastDmxUpdate Outputs/.stDMXOutDataLinie01/arrData @bit 3384 <-> DMX Channel 385-448/Channel 424
//     FastDmxUpdate Outputs/.stDMXOutDataLinie01/arrData @bit 3392 <-> DMX Channel 385-448/Channel 425
//     FastDmxUpdate Outputs/.stDMXOutDataLinie01/arrData @bit 3400 <-> DMX Channel 385-448/Channel 426
//     FastDmxUpdate Outputs/.stDMXOutDataLinie01/arrData @bit 3408 <-> DMX Channel 385-448/Channel 427
//     FastDmxUpdate Outputs/.stDMXOutDataLinie01/arrData @bit 3416 <-> DMX Channel 385-448/Channel 428
//     FastDmxUpdate Outputs/.stDMXOutDataLinie01/arrData @bit 3424 <-> DMX Channel 385-448/Channel 429
//     FastDmxUpdate Outputs/.stDMXOutDataLinie01/arrData @bit 3432 <-> DMX Channel 385-448/Channel 430
//     FastDmxUpdate Outputs/.stDMXOutDataLinie01/arrData @bit 3440 <-> DMX Channel 385-448/Channel 431
//     FastDmxUpdate Outputs/.stDMXOutDataLinie01/arrData @bit 3448 <-> DMX Channel 385-448/Channel 432
//     FastDmxUpdate Outputs/.stDMXOutDataLinie01/arrData @bit 3456 <-> DMX Channel 385-448/Channel 433
//     FastDmxUpdate Outputs/.stDMXOutDataLinie01/arrData @bit 3464 <-> DMX Channel 385-448/Channel 434
//     FastDmxUpdate Outputs/.stDMXOutDataLinie01/arrData @bit 3472 <-> DMX Channel 385-448/Channel 435
//     FastDmxUpdate Outputs/.stDMXOutDataLinie01/arrData @bit 3480 <-> DMX Channel 385-448/Channel 436
//     FastDmxUpdate Outputs/.stDMXOutDataLinie01/arrData @bit 3488 <-> DMX Channel 385-448/Channel 437
//     FastDmxUpdate Outputs/.stDMXOutDataLinie01/arrData @bit 3496 <-> DMX Channel 385-448/Channel 438
//     FastDmxUpdate Outputs/.stDMXOutDataLinie01/arrData @bit 3504 <-> DMX Channel 385-448/Channel 439
//     FastDmxUpdate Outputs/.stDMXOutDataLinie01/arrData @bit 3512 <-> DMX Channel 385-448/Channel 440
//     FastDmxUpdate Outputs/.stDMXOutDataLinie01/arrData @bit 3520 <-> DMX Channel 385-448/Channel 441
//     FastDmxUpdate Outputs/.stDMXOutDataLinie01/arrData @bit 3528 <-> DMX Channel 385-448/Channel 442
//     FastDmxUpdate Outputs/.stDMXOutDataLinie01/arrData @bit 3536 <-> DMX Channel 385-448/Channel 443
//     FastDmxUpdate Outputs/.stDMXOutDataLinie01/arrData @bit 3544 <-> DMX Channel 385-448/Channel 444
//     FastDmxUpdate Outputs/.stDMXOutDataLinie01/arrData @bit 3552 <-> DMX Channel 385-448/Channel 445
//     FastDmxUpdate Outputs/.stDMXOutDataLinie01/arrData @bit 3560 <-> DMX Channel 385-448/Channel 446
//     FastDmxUpdate Outputs/.stDMXOutDataLinie01/arrData @bit 3568 <-> DMX Channel 385-448/Channel 447
//     FastDmxUpdate Outputs/.stDMXOutDataLinie01/arrData @bit 3576 <-> DMX Channel 385-448/Channel 448
//     FastDmxUpdate Outputs/.stDMXOutDataLinie01/arrData @bit 3584 <-> DMX Channel 449-512/Channel 449
//     FastDmxUpdate Outputs/.stDMXOutDataLinie01/arrData @bit 3592 <-> DMX Channel 449-512/Channel 450
//     FastDmxUpdate Outputs/.stDMXOutDataLinie01/arrData @bit 3600 <-> DMX Channel 449-512/Channel 451
//     FastDmxUpdate Outputs/.stDMXOutDataLinie01/arrData @bit 3608 <-> DMX Channel 449-512/Channel 452
//     FastDmxUpdate Outputs/.stDMXOutDataLinie01/arrData @bit 3616 <-> DMX Channel 449-512/Channel 453
//     FastDmxUpdate Outputs/.stDMXOutDataLinie01/arrData @bit 3624 <-> DMX Channel 449-512/Channel 454
//     FastDmxUpdate Outputs/.stDMXOutDataLinie01/arrData @bit 3632 <-> DMX Channel 449-512/Channel 455
//     FastDmxUpdate Outputs/.stDMXOutDataLinie01/arrData @bit 3640 <-> DMX Channel 449-512/Channel 456
//     FastDmxUpdate Outputs/.stDMXOutDataLinie01/arrData @bit 3648 <-> DMX Channel 449-512/Channel 457
//     FastDmxUpdate Outputs/.stDMXOutDataLinie01/arrData @bit 3656 <-> DMX Channel 449-512/Channel 458
//     FastDmxUpdate Outputs/.stDMXOutDataLinie01/arrData @bit 3664 <-> DMX Channel 449-512/Channel 459
//     FastDmxUpdate Outputs/.stDMXOutDataLinie01/arrData @bit 3672 <-> DMX Channel 449-512/Channel 460
//     FastDmxUpdate Outputs/.stDMXOutDataLinie01/arrData @bit 3680 <-> DMX Channel 449-512/Channel 461
//     FastDmxUpdate Outputs/.stDMXOutDataLinie01/arrData @bit 3688 <-> DMX Channel 449-512/Channel 462
//     FastDmxUpdate Outputs/.stDMXOutDataLinie01/arrData @bit 3696 <-> DMX Channel 449-512/Channel 463
//     FastDmxUpdate Outputs/.stDMXOutDataLinie01/arrData @bit 3704 <-> DMX Channel 449-512/Channel 464
//     FastDmxUpdate Outputs/.stDMXOutDataLinie01/arrData @bit 3712 <-> DMX Channel 449-512/Channel 465
//     FastDmxUpdate Outputs/.stDMXOutDataLinie01/arrData @bit 3720 <-> DMX Channel 449-512/Channel 466
//     FastDmxUpdate Outputs/.stDMXOutDataLinie01/arrData @bit 3728 <-> DMX Channel 449-512/Channel 467
//     FastDmxUpdate Outputs/.stDMXOutDataLinie01/arrData @bit 3736 <-> DMX Channel 449-512/Channel 468
//     FastDmxUpdate Outputs/.stDMXOutDataLinie01/arrData @bit 3744 <-> DMX Channel 449-512/Channel 469
//     FastDmxUpdate Outputs/.stDMXOutDataLinie01/arrData @bit 3752 <-> DMX Channel 449-512/Channel 470
//     FastDmxUpdate Outputs/.stDMXOutDataLinie01/arrData @bit 3760 <-> DMX Channel 449-512/Channel 471
//     FastDmxUpdate Outputs/.stDMXOutDataLinie01/arrData @bit 3768 <-> DMX Channel 449-512/Channel 472
//     FastDmxUpdate Outputs/.stDMXOutDataLinie01/arrData @bit 3776 <-> DMX Channel 449-512/Channel 473
//     FastDmxUpdate Outputs/.stDMXOutDataLinie01/arrData @bit 3784 <-> DMX Channel 449-512/Channel 474
//     FastDmxUpdate Outputs/.stDMXOutDataLinie01/arrData @bit 3792 <-> DMX Channel 449-512/Channel 475
//     FastDmxUpdate Outputs/.stDMXOutDataLinie01/arrData @bit 3800 <-> DMX Channel 449-512/Channel 476
//     FastDmxUpdate Outputs/.stDMXOutDataLinie01/arrData @bit 3808 <-> DMX Channel 449-512/Channel 477
//     FastDmxUpdate Outputs/.stDMXOutDataLinie01/arrData @bit 3816 <-> DMX Channel 449-512/Channel 478
//     FastDmxUpdate Outputs/.stDMXOutDataLinie01/arrData @bit 3824 <-> DMX Channel 449-512/Channel 479
//     FastDmxUpdate Outputs/.stDMXOutDataLinie01/arrData @bit 3832 <-> DMX Channel 449-512/Channel 480
//     FastDmxUpdate Outputs/.stDMXOutDataLinie01/arrData @bit 3840 <-> DMX Channel 449-512/Channel 481
//     FastDmxUpdate Outputs/.stDMXOutDataLinie01/arrData @bit 3848 <-> DMX Channel 449-512/Channel 482
//     FastDmxUpdate Outputs/.stDMXOutDataLinie01/arrData @bit 3856 <-> DMX Channel 449-512/Channel 483
//     FastDmxUpdate Outputs/.stDMXOutDataLinie01/arrData @bit 3864 <-> DMX Channel 449-512/Channel 484
//     FastDmxUpdate Outputs/.stDMXOutDataLinie01/arrData @bit 3872 <-> DMX Channel 449-512/Channel 485
//     FastDmxUpdate Outputs/.stDMXOutDataLinie01/arrData @bit 3880 <-> DMX Channel 449-512/Channel 486
//     FastDmxUpdate Outputs/.stDMXOutDataLinie01/arrData @bit 3888 <-> DMX Channel 449-512/Channel 487
//     FastDmxUpdate Outputs/.stDMXOutDataLinie01/arrData @bit 3896 <-> DMX Channel 449-512/Channel 488
//     FastDmxUpdate Outputs/.stDMXOutDataLinie01/arrData @bit 3904 <-> DMX Channel 449-512/Channel 489
//     FastDmxUpdate Outputs/.stDMXOutDataLinie01/arrData @bit 3912 <-> DMX Channel 449-512/Channel 490
//     FastDmxUpdate Outputs/.stDMXOutDataLinie01/arrData @bit 3920 <-> DMX Channel 449-512/Channel 491
//     FastDmxUpdate Outputs/.stDMXOutDataLinie01/arrData @bit 3928 <-> DMX Channel 449-512/Channel 492
//     FastDmxUpdate Outputs/.stDMXOutDataLinie01/arrData @bit 3936 <-> DMX Channel 449-512/Channel 493
//     FastDmxUpdate Outputs/.stDMXOutDataLinie01/arrData @bit 3944 <-> DMX Channel 449-512/Channel 494
//     FastDmxUpdate Outputs/.stDMXOutDataLinie01/arrData @bit 3952 <-> DMX Channel 449-512/Channel 495
//     FastDmxUpdate Outputs/.stDMXOutDataLinie01/arrData @bit 3960 <-> DMX Channel 449-512/Channel 496
//     FastDmxUpdate Outputs/.stDMXOutDataLinie01/arrData @bit 3968 <-> DMX Channel 449-512/Channel 497
//     FastDmxUpdate Outputs/.stDMXOutDataLinie01/arrData @bit 3976 <-> DMX Channel 449-512/Channel 498
//     FastDmxUpdate Outputs/.stDMXOutDataLinie01/arrData @bit 3984 <-> DMX Channel 449-512/Channel 499
//     FastDmxUpdate Outputs/.stDMXOutDataLinie01/arrData @bit 3992 <-> DMX Channel 449-512/Channel 500
//     FastDmxUpdate Outputs/.stDMXOutDataLinie01/arrData @bit 4000 <-> DMX Channel 449-512/Channel 501
//     FastDmxUpdate Outputs/.stDMXOutDataLinie01/arrData @bit 4008 <-> DMX Channel 449-512/Channel 502
//     FastDmxUpdate Outputs/.stDMXOutDataLinie01/arrData @bit 4016 <-> DMX Channel 449-512/Channel 503
//     FastDmxUpdate Outputs/.stDMXOutDataLinie01/arrData @bit 4024 <-> DMX Channel 449-512/Channel 504
//     FastDmxUpdate Outputs/.stDMXOutDataLinie01/arrData @bit 4032 <-> DMX Channel 449-512/Channel 505
//     FastDmxUpdate Outputs/.stDMXOutDataLinie01/arrData @bit 4040 <-> DMX Channel 449-512/Channel 506
//     FastDmxUpdate Outputs/.stDMXOutDataLinie01/arrData @bit 4048 <-> DMX Channel 449-512/Channel 507
//     FastDmxUpdate Outputs/.stDMXOutDataLinie01/arrData @bit 4056 <-> DMX Channel 449-512/Channel 508
//     FastDmxUpdate Outputs/.stDMXOutDataLinie01/arrData @bit 4064 <-> DMX Channel 449-512/Channel 509
//     FastDmxUpdate Outputs/.stDMXOutDataLinie01/arrData @bit 4072 <-> DMX Channel 449-512/Channel 510
//     FastDmxUpdate Outputs/.stDMXOutDataLinie01/arrData @bit 4080 <-> DMX Channel 449-512/Channel 511
//     FastDmxUpdate Outputs/.stDMXOutDataLinie01/arrData @bit 4088 <-> DMX Channel 449-512/Channel 512
//     FastDmxUpdate Outputs/.stDMXOutDataLinie01/arrData @bit 792 <-> DMX Channel 65-128/Channel 100
//     FastDmxUpdate Outputs/.stDMXOutDataLinie01/arrData @bit 800 <-> DMX Channel 65-128/Channel 101
//     FastDmxUpdate Outputs/.stDMXOutDataLinie01/arrData @bit 808 <-> DMX Channel 65-128/Channel 102
//     FastDmxUpdate Outputs/.stDMXOutDataLinie01/arrData @bit 816 <-> DMX Channel 65-128/Channel 103
//     FastDmxUpdate Outputs/.stDMXOutDataLinie01/arrData @bit 824 <-> DMX Channel 65-128/Channel 104
//     FastDmxUpdate Outputs/.stDMXOutDataLinie01/arrData @bit 832 <-> DMX Channel 65-128/Channel 105
//     FastDmxUpdate Outputs/.stDMXOutDataLinie01/arrData @bit 840 <-> DMX Channel 65-128/Channel 106
//     FastDmxUpdate Outputs/.stDMXOutDataLinie01/arrData @bit 848 <-> DMX Channel 65-128/Channel 107
//     FastDmxUpdate Outputs/.stDMXOutDataLinie01/arrData @bit 856 <-> DMX Channel 65-128/Channel 108
//     FastDmxUpdate Outputs/.stDMXOutDataLinie01/arrData @bit 864 <-> DMX Channel 65-128/Channel 109
//     FastDmxUpdate Outputs/.stDMXOutDataLinie01/arrData @bit 872 <-> DMX Channel 65-128/Channel 110
//     FastDmxUpdate Outputs/.stDMXOutDataLinie01/arrData @bit 880 <-> DMX Channel 65-128/Channel 111
//     FastDmxUpdate Outputs/.stDMXOutDataLinie01/arrData @bit 888 <-> DMX Channel 65-128/Channel 112
//     FastDmxUpdate Outputs/.stDMXOutDataLinie01/arrData @bit 896 <-> DMX Channel 65-128/Channel 113
//     FastDmxUpdate Outputs/.stDMXOutDataLinie01/arrData @bit 904 <-> DMX Channel 65-128/Channel 114
//     FastDmxUpdate Outputs/.stDMXOutDataLinie01/arrData @bit 912 <-> DMX Channel 65-128/Channel 115
//     FastDmxUpdate Outputs/.stDMXOutDataLinie01/arrData @bit 920 <-> DMX Channel 65-128/Channel 116
//     FastDmxUpdate Outputs/.stDMXOutDataLinie01/arrData @bit 928 <-> DMX Channel 65-128/Channel 117
//     FastDmxUpdate Outputs/.stDMXOutDataLinie01/arrData @bit 936 <-> DMX Channel 65-128/Channel 118
//     FastDmxUpdate Outputs/.stDMXOutDataLinie01/arrData @bit 944 <-> DMX Channel 65-128/Channel 119
//     FastDmxUpdate Outputs/.stDMXOutDataLinie01/arrData @bit 952 <-> DMX Channel 65-128/Channel 120
//     FastDmxUpdate Outputs/.stDMXOutDataLinie01/arrData @bit 960 <-> DMX Channel 65-128/Channel 121
//     FastDmxUpdate Outputs/.stDMXOutDataLinie01/arrData @bit 968 <-> DMX Channel 65-128/Channel 122
//     FastDmxUpdate Outputs/.stDMXOutDataLinie01/arrData @bit 976 <-> DMX Channel 65-128/Channel 123
//     FastDmxUpdate Outputs/.stDMXOutDataLinie01/arrData @bit 984 <-> DMX Channel 65-128/Channel 124
//     FastDmxUpdate Outputs/.stDMXOutDataLinie01/arrData @bit 992 <-> DMX Channel 65-128/Channel 125
//     FastDmxUpdate Outputs/.stDMXOutDataLinie01/arrData @bit 1000 <-> DMX Channel 65-128/Channel 126
//     FastDmxUpdate Outputs/.stDMXOutDataLinie01/arrData @bit 1008 <-> DMX Channel 65-128/Channel 127
//     FastDmxUpdate Outputs/.stDMXOutDataLinie01/arrData @bit 1016 <-> DMX Channel 65-128/Channel 128
//     FastDmxUpdate Outputs/.stDMXOutDataLinie01/arrData @bit 512 <-> DMX Channel 65-128/Channel 65
//     FastDmxUpdate Outputs/.stDMXOutDataLinie01/arrData @bit 520 <-> DMX Channel 65-128/Channel 66
//     FastDmxUpdate Outputs/.stDMXOutDataLinie01/arrData @bit 528 <-> DMX Channel 65-128/Channel 67
//     FastDmxUpdate Outputs/.stDMXOutDataLinie01/arrData @bit 536 <-> DMX Channel 65-128/Channel 68
//     FastDmxUpdate Outputs/.stDMXOutDataLinie01/arrData @bit 544 <-> DMX Channel 65-128/Channel 69
//     FastDmxUpdate Outputs/.stDMXOutDataLinie01/arrData @bit 552 <-> DMX Channel 65-128/Channel 70
//     FastDmxUpdate Outputs/.stDMXOutDataLinie01/arrData @bit 560 <-> DMX Channel 65-128/Channel 71
//     FastDmxUpdate Outputs/.stDMXOutDataLinie01/arrData @bit 568 <-> DMX Channel 65-128/Channel 72
//     FastDmxUpdate Outputs/.stDMXOutDataLinie01/arrData @bit 576 <-> DMX Channel 65-128/Channel 73
//     FastDmxUpdate Outputs/.stDMXOutDataLinie01/arrData @bit 584 <-> DMX Channel 65-128/Channel 74
//     FastDmxUpdate Outputs/.stDMXOutDataLinie01/arrData @bit 592 <-> DMX Channel 65-128/Channel 75
//     FastDmxUpdate Outputs/.stDMXOutDataLinie01/arrData @bit 600 <-> DMX Channel 65-128/Channel 76
//     FastDmxUpdate Outputs/.stDMXOutDataLinie01/arrData @bit 608 <-> DMX Channel 65-128/Channel 77
//     FastDmxUpdate Outputs/.stDMXOutDataLinie01/arrData @bit 616 <-> DMX Channel 65-128/Channel 78
//     FastDmxUpdate Outputs/.stDMXOutDataLinie01/arrData @bit 624 <-> DMX Channel 65-128/Channel 79
//     FastDmxUpdate Outputs/.stDMXOutDataLinie01/arrData @bit 632 <-> DMX Channel 65-128/Channel 80
//     FastDmxUpdate Outputs/.stDMXOutDataLinie01/arrData @bit 640 <-> DMX Channel 65-128/Channel 81
//     FastDmxUpdate Outputs/.stDMXOutDataLinie01/arrData @bit 648 <-> DMX Channel 65-128/Channel 82
//     FastDmxUpdate Outputs/.stDMXOutDataLinie01/arrData @bit 656 <-> DMX Channel 65-128/Channel 83
//     FastDmxUpdate Outputs/.stDMXOutDataLinie01/arrData @bit 664 <-> DMX Channel 65-128/Channel 84
//     FastDmxUpdate Outputs/.stDMXOutDataLinie01/arrData @bit 672 <-> DMX Channel 65-128/Channel 85
//     FastDmxUpdate Outputs/.stDMXOutDataLinie01/arrData @bit 680 <-> DMX Channel 65-128/Channel 86
//     FastDmxUpdate Outputs/.stDMXOutDataLinie01/arrData @bit 688 <-> DMX Channel 65-128/Channel 87
//     FastDmxUpdate Outputs/.stDMXOutDataLinie01/arrData @bit 696 <-> DMX Channel 65-128/Channel 88
//     FastDmxUpdate Outputs/.stDMXOutDataLinie01/arrData @bit 704 <-> DMX Channel 65-128/Channel 89
//     FastDmxUpdate Outputs/.stDMXOutDataLinie01/arrData @bit 712 <-> DMX Channel 65-128/Channel 90
//     FastDmxUpdate Outputs/.stDMXOutDataLinie01/arrData @bit 720 <-> DMX Channel 65-128/Channel 91
//     FastDmxUpdate Outputs/.stDMXOutDataLinie01/arrData @bit 728 <-> DMX Channel 65-128/Channel 92
//     FastDmxUpdate Outputs/.stDMXOutDataLinie01/arrData @bit 736 <-> DMX Channel 65-128/Channel 93
//     FastDmxUpdate Outputs/.stDMXOutDataLinie01/arrData @bit 744 <-> DMX Channel 65-128/Channel 94
//     FastDmxUpdate Outputs/.stDMXOutDataLinie01/arrData @bit 752 <-> DMX Channel 65-128/Channel 95
//     FastDmxUpdate Outputs/.stDMXOutDataLinie01/arrData @bit 760 <-> DMX Channel 65-128/Channel 96
//     FastDmxUpdate Outputs/.stDMXOutDataLinie01/arrData @bit 768 <-> DMX Channel 65-128/Channel 97
//     FastDmxUpdate Outputs/.stDMXOutDataLinie01/arrData @bit 776 <-> DMX Channel 65-128/Channel 98
//     FastDmxUpdate Outputs/.stDMXOutDataLinie01/arrData @bit 784 <-> DMX Channel 65-128/Channel 99
//     FastDmxUpdate Outputs/.stDMXOutDataLinie01/bDisableCyclicTxD <-> DMX Control/Disable cyclic TxD
//     FastDmxUpdate Outputs/.stDMXOutDataLinie01/bSendDefaultData <-> DMX Control/Send default data
//     FastDmxUpdate Outputs/.stDMXOutDataLinie01/bTransmitRequest <-> DMX Control/Transmit request
//     FastDmxUpdate Outputs/.stDMXOutDataLinie01/byStartCode <-> DMX Control/Start code
//     FastDmxUpdate Outputs/.stDMXOutDataLinie01/wChannelLength <-> DMX Control/Channel length
//   BAUK_EK_BMS_PLC/BAUK_EK_BMS_PLC Instance <-> CX2040 E-Bus/CX2040 Supply/Server Room EtherCAT Junction/OLD BLIND CONTROL/Blind Control Boardroom
//     PlcTask Inputs/BackgroundComms.HubCommIn[2]/D <-> COM Inputs/Data In 0
//     PlcTask Inputs/BackgroundComms.HubCommIn[2]/D @bit {8..168 step 8} <-> COM Inputs/Data In {1..21}  (21 links)
//     PlcTask Inputs/BackgroundComms.HubCommIn[2]/Status <-> COM Inputs/Status
//     PlcTask Outputs/BackgroundComms.HubCommOut[2]/Ctrl <-> COM Outputs/Ctrl
//     PlcTask Outputs/BackgroundComms.HubCommOut[2]/D <-> COM Outputs/Data Out 0
//     PlcTask Outputs/BackgroundComms.HubCommOut[2]/D @bit {8..168 step 8} <-> COM Outputs/Data Out {1..21}  (21 links)
//   BAUK_EK_BMS_PLC/BAUK_EK_BMS_PLC Instance <-> CX2040 E-Bus/CX2040 Supply/Server Room EtherCAT Junction/OLD BLIND CONTROL/Blind Control Communal Area
//     PlcTask Inputs/BackgroundComms.HubCommIn[1]/D <-> COM Inputs/Data In 0
//     PlcTask Inputs/BackgroundComms.HubCommIn[1]/D @bit {8..168 step 8} <-> COM Inputs/Data In {1..21}  (21 links)
//     PlcTask Inputs/BackgroundComms.HubCommIn[1]/Status <-> COM Inputs/Status
//     PlcTask Outputs/BackgroundComms.HubCommOut[1]/Ctrl <-> COM Outputs/Ctrl
//     PlcTask Outputs/BackgroundComms.HubCommOut[1]/D <-> COM Outputs/Data Out 0
//     PlcTask Outputs/BackgroundComms.HubCommOut[1]/D @bit {8..168 step 8} <-> COM Outputs/Data Out {1..21}  (21 links)
//   BAUK_EK_BMS_PLC/BAUK_EK_BMS_PLC Instance <-> CX2040 E-Bus/CX2040 Supply/Server Room EtherCAT Junction/OLD BLIND CONTROL/Blind Control Staff Room
//     PlcTask Inputs/BackgroundComms.HubCommIn[0]/D <-> COM Inputs/Data In 0
//     PlcTask Inputs/BackgroundComms.HubCommIn[0]/D @bit {8..168 step 8} <-> COM Inputs/Data In {1..21}  (21 links)
//     PlcTask Inputs/BackgroundComms.HubCommIn[0]/Status <-> COM Inputs/Status
//     PlcTask Outputs/BackgroundComms.HubCommOut[0]/Ctrl <-> COM Outputs/Ctrl
//     PlcTask Outputs/BackgroundComms.HubCommOut[0]/D <-> COM Outputs/Data Out 0
//     PlcTask Outputs/BackgroundComms.HubCommOut[0]/D @bit {8..168 step 8} <-> COM Outputs/Data Out {1..21}  (21 links)
//   BAUK_EK_BMS_PLC/BAUK_EK_BMS_PLC Instance <-> CX2040 E-Bus/CX2040 Supply/Server Room EtherCAT Junction/OLD BLIND CONTROL/Coffee Machine Power Monitor
//     PlcTask Inputs/.diActivePower <-> PM Inputs Channel 1/Active power
//     PlcTask Inputs/.diCurrent <-> PM Inputs Channel 1/Current
//     PlcTask Inputs/.diVarientValue <-> PM Inputs Channel 1/Variant value
//     PlcTask Inputs/.diVoltage <-> PM Inputs Channel 1/Voltage
//     PlcTask Inputs/.uiPresentIndex <-> PM Inputs Channel 1/Index
//     PlcTask Outputs/.uiIndexRequest <-> PM Outputs Channel 1/Index

CONFIGURATION BAUK_EK_BMS_PLC
    RESOURCE PLC ON TwinCAT3
        TASK FastDmxUpdate(INTERVAL := T#1ms, PRIORITY := 1);
        PROGRAM DMX WITH FastDmxUpdate : DMX;
    END_RESOURCE
END_CONFIGURATION

// ---- HMI/TIMESTR_Strings.TcDUT
TYPE TIMESTR_Strings :
STRUCT
	sYear: STRING;
	sMonth: STRING;
	sDayOfWeek: STRING;
	sDay: STRING;
	sHour: STRING;
	sMinute: STRING;
	sSecond: STRING;
	sMillisecond: STRING;
END_STRUCT
END_TYPE

// ---- LIGHTS/DMX/ST_RGB.TcDUT
TYPE ST_RGB :
STRUCT
	red		:	BYTE;
	green	:	BYTE;
	blue	:	BYTE;
END_STRUCT
END_TYPE

// ---- POWER MONITORING/ST_EL3403_Data.TcDUT
TYPE ST_EL3403_Data :
STRUCT
	current			:	REAL; 	// 0.000001 A
	voltage			:	REAL; 	// 0.0001 V
	activePower		:	REAL;	// 0.01 W
	apparentPower	:	REAL;	// 0.01 VA
	reactivePower	:	REAL;	// 0.01 VAR
	positiveEnergy	:	REAL;	// 0.001 Wh
	cosPhi			:	REAL;	// 0.001
	frequency		:	REAL;	// 0.1 Hz
	negativeEnergy	:	REAL;	// 0.001 Wh
END_STRUCT
END_TYPE

// ---- WORKSHOP WALL/ST_PsuDiagData.TcDUT
{attribute 'pack_mode' := '1'}
TYPE ST_PsuDiagData :
STRUCT
	{attribute 'hide'}
	align1						:	UINT;
	minInputVoltage				:	REAL; //V
	inputUnderVoltageCounter	:	UINT;
	maxInputVoltage				:	REAL; //V
	{attribute 'hide'}
	align2						:	UINT;
	maxPeakInputVoltage			:	REAL; //V
	inputOvervoltageCounter		:	UINT;
	minTemperature				:	REAL; //°C
	maxTemperature				:	REAL; //°C
	actualRMSInputVoltage		:	REAL; //V
	{attribute 'hide'}
	align3						:	UDINT;
	actualTemperature			:	REAL; //°C
END_STRUCT
END_TYPE

// ---- WORKSHOP WALL/ST_PsuInfoData.TcDUT
{attribute 'pack_mode' := '1'}
TYPE ST_PsuInfoData :
STRUCT
	{attribute 'hide'}
	align1			:	UDINT;
	{attribute 'hide'}
	align2			:	UINT;
	operatingTime	:	UDINT; // seconds
	upTime			:	UDINT; // seconds
	turnOnCounter	:	UDINT;
	{attribute 'hide'}
	align3			:	UINT;
END_STRUCT
END_TYPE

// ---- Global_Variables.TcGVL
{attribute 'Tc2GvlVarNames'}
VAR_GLOBAL
	///Current Table Shown on main page
	BlankCurrentMonthSignInTable			: 	ARRAY[0..nMaxTableLength] OF ST_SignInTable;
	///Visulization             			  	
	sVisuName								: 	STRING(255);
	sVisuCompany							: 	STRING(255);
	sVisuPersonVisiting						: 	STRING(255);
	sVisuReason								: 	STRING(255);
	sVisuVehicleReg							: 	STRING(10);
	sVisusDateIn							: 	STRING(8);
	sVisusTimeIn							: 	STRING(8);
	
	
	///Visu Variables
	xVisuSignInButton						: 	BOOL;
	xVisuSignOutButton						: 	BOOL;
	xVisuHideSignInButton					: 	BOOL;
	xVisuYesPCControl						: 	BOOL;
	nVisuTableRowSelection					: 	INT;
	nVisuTableColumnSelection				: 	INT;
	sVisuEmailAddress						: 	STRING;
	///Date Time Variables
	STDateTimeStrings						: 	TIMESTR_Strings;
	sDate									: 	STRING;
	sTime									:	STRING;
	
	ComboBoxCurrentMonthSignInTable 		: 	ARRAY[0..nMaxTableLength] OF STRING;
	BlankComboBoxCurrentMonthSignInTable	: 	ARRAY[0..nMaxTableLength] OF STRING;
	
	test : STRING;
	
	numberOfOpenWindows				AT%Q* 	:	WORD;
	boardroomModeIsProjector		AT%Q* 	:	BOOL;
	boardroomModeIsFullOn			AT%Q* 	:	BOOL;
	setBoardroomGold				AT%I* 	:	BOOL;
	setBoardroomPurple				AT%I* 	:	BOOL;
	setBoardroomRed					AT%I* 	:	BOOL;
	communalLux1					AT%Q* 	: 	INT;
	communalLux2					AT%Q* 	: 	INT;
	communalOccupancy1				AT%Q* 	: 	BOOL;
	communalOccupancy2				AT%Q* 	: 	BOOL;
	staffLux1						AT%Q* 	: 	INT;
	staffLux2						AT%Q* 	: 	INT;
	staffOccupancy1					AT%Q* 	: 	BOOL;
	staffOccupancy2					AT%Q* 	: 	BOOL;
	boardLux1						AT%Q* 	: 	INT;
	boardLux2						AT%Q* 	: 	INT;
	boardOccupancy1					AT%Q* 	: 	BOOL;
	boardOccupancy2					AT%Q* 	: 	BOOL;
	//Enocean Socket Control Bits

	xXplanarScreenPowerOn					:	BOOL;
	xXplanarScreenPowerOff					:	BOOL;
	
	xSleepMode								:	BOOL;

	EnOceanComms							: 	STR_KL6581;

	stKL6581InData 					AT%I*	:	KL6581_Input;
	stKL6581OutData 				AT%Q*	:	KL6581_Output;

	stCommandBuffer 						: 	ST_DALIV2CommandBuffer;

	stDALIInData    				AT%I*	: 	ST_DALIV2InData;
	stDALIOutData  					AT%Q*	: 	ST_DALIV2OutData;
	
	stKL6811InData    				AT%I*	: 	Tc3_DALI.ST_KL6811InData;
	stKL6811OutData  				AT%Q*	: 	Tc3_DALI.ST_KL6811OutData;

	(* DMX Line *)
	stDMXInDataLinie01              AT%I*	:	ST_EL6851InData;
	stDMXOutDataLinie01             AT%Q*	:	ST_EL6851OutData;
	stCommandBuffer01						:	ST_DMXCommandBuffer;
	
	arrDMXProcessData						:	ARRAY [1..512] 	OF BYTE;
	FBEnOceanPTM200							:	ARRAY [0..3] 	OF FB_EnOceanPTM200; 
	FBEnOceanSTM250							:	ARRAY [0..5] 	OF FB_EnOceanSTM250;
		
	EnoceanTransmitterID					: 	ARRAY [0..3] 	OF UDINT := [3035027, 3030651, 3036382, 3030640];
	EnoceanTransmitterIDWindows				: 	ARRAY [0..5] 	OF UDINT := [85424832, 85423614, 93313507, 85423331, 85423280, 85423273]; 
	
	PTM200StrippedTables					:	ARRAY [0..15] 	OF SwitchTable;
	PTM250WindowSensor						:	ARRAY [0..5]	OF BOOL;
	
	FBDALIV2Light							:	ARRAY [0..57] 	OF FB_DALIV2Light;
	FBDALIV2QueryLightState					:	ARRAY [0..57] 	OF FB_DALIV2QueryLampPowerOn;
	tLightTable								:	ARRAY [0..57] 	OF LightTable;
	
	BlindCX7000UserTable					: 	ARRAY [0..2] 	OF StructBlindControl := [(JogTimeInt:=3000)];
	BlindCommandTable 				AT%MB0	:	ARRAY [0..19] 	OF UINT;		

	CP67BoardRoomLightsOn			AT%MB40	:	BYTE;
	BoardroomActualLightLvl 		AT%MB42	:	BYTE;
	
	
	AWindowIsOpenLightTrigger				:	BOOL;
	
	diPh1Voltage							:	DINT;
	diPh1Current							:	DINT;
	diPh1ActivePower						:	DINT;

	diVoltage						AT%IB0	:	DINT;
	diCurrent						AT%IB4	:	DINT;
	diActivePower					AT%IB8	:	DINT;
	diFrequency						AT%IB12	:	DINT;
	diVarientValue					AT%IB16	:	DINT;
	uiPresentIndex					AT%IB20	:	USINT;
	uiIndexRequest					AT%QB17	:	USINT := 4;

	Mains_Varient_Raw						: 	ARRAY [0..6] OF DINT;

	VisuGroupSelect							:	INT;

	AdvancedBlindControl					:	ARRAY [1..16] OF StructAdvancedBlindControl;


	PassADSBlindInfo				AT %MB0	:	ARRAY [0..19] OF UINT;

	PassADSBlindControlCP67					:	ARRAY [1..57] OF BYTE;


	(* Blind Modes/Scenes*)

	BoardRoom_PrivacyMode					:	BOOL;
	BoardRoom_SceneryMode					:	BOOL;
	BoardRoom_ProjectorMode					:	BOOL;
	BoardRoom_MeetingMode					:	BOOL;
                                			
	DeskArea_PrivacyMode					:	BOOL;
	DeskArea_SceneryMode					:	BOOL;
	DeskArea_NightMode						:	BOOL;
	DeskArea_MorningMode					:	BOOL;
                                			    
	KitchenArea_PrivacyMode					:	BOOL;
	KitchenArea_SceneryMode					:	BOOL;
	KitchenArea_NightMode					:	BOOL;
	KitchenArea_MorningMode					:	BOOL;
                                	            
	EntireBuilding_CleaningMode				:	BOOL;
	
	(* Wind Turbine Data*)
	WindSpeed						AT%M*	:	LREAL;
	RPM								AT%M*	:	LREAL;
	Power							AT%M*	:	LREAL;
	
	(* Blind Stretch*)
	BlindSelector					AT%M*	:	INT;

END_VAR

VAR_GLOBAL CONSTANT
	BUFFER_SIZE								: 	INT := 10000;
	nMaxTableLength							: 	INT := 50;
END_VAR


VAR_GLOBAL PERSISTENT
	CurrentMonthSignInTable					: 	ARRAY[0..nMaxTableLength] OF ST_SignInTable;
	KWAccumulate							:	REAL;
	KWHReading								:	REAL;
	Cost									:	REAL;

END_VAR

// ---- LIGHTS/DMX/DMX.TcPOU
PROGRAM DMX
VAR
	fbEL6851Communication	:	FB_EL6851Communication;

	byTopLeftShelfRed		: BYTE;                                   
	byTopLeftShelfGreen		: BYTE;                                   
	byTopLeftShelfBlue		: BYTE;                                   
	byMiddle1LeftShelfRed	: BYTE;                                   
	byMiddle1LeftShelfGreen	: BYTE;	                               
	byMiddle1LeftShelfBlue	: BYTE;	                               
	byMiddle2LeftShelfRed	: BYTE;	                               
	byMiddle2LeftShelfGreen	: BYTE;                                  
	byMiddle2LeftShelfBlue	: BYTE;	                               
	byBottomLeftShelfRed	: BYTE;                                   
	byBottomLeftShelfGreen	: BYTE;                                   
	byBottomLeftShelfBlue	: BYTE;                                   
	byTopRightShelfRed		: BYTE;                                   
	byTopRightShelfGreen	: BYTE;                                   
	byTopRightShelfBlue		: BYTE;	                               
	byMiddle1RightShelfRed	: BYTE;	                               
	byMiddle1RightShelfGreen: BYTE;                                   
	byMiddle1RightShelfBlue	: BYTE;                                  
	byMiddle2RightShelfRed	: BYTE;                                   
	byMiddle2RightShelfGreen: BYTE;                                   
	byMiddle2RightShelfBlue	: BYTE;                                   
	byBottomRightShelfRed	: BYTE;                                   
	byBottomRightShelfGreen	: BYTE;                                   
	byBottomRightShelfBlue	: BYTE;

	colours					:	ST_RGB; //Used for HMI colour picker interaction
	shelfSelection			:	ARRAY [1..8] OF BOOL;
	hmiUpdateTimer			:	Pulse;
	updateHmi				:	BOOL;
END_VAR

//DMX Handle
fbEL6851Communication(wSourceManufacturerID := 16#42_41,
						dwSourceDeviceID := 16#12_13_14_15,
						bEnableSendingData := TRUE,
						bSetCycleMode := TRUE,
						bSendDefaultData := FALSE,
						uiDataLength := 512,
						dwOptions := 0,
						stEL6851InData := stDMXInDataLinie01,
						stEL6851OutData := stDMXOutDataLinie01,
						stCommandBuffer := stCommandBuffer01,
						arrProcessData := arrDMXProcessData);

//Update RGB DMX process data
MoveDMXValues();					
	
	IF FBEnOceanPTM200[2].bSwitches[0] THEN
		byTopLeftShelfRed			 := 254;
		byMiddle1LeftShelfRed		 := 254;	 
		byMiddle2LeftShelfRed		 := 254;	
		byBottomLeftShelfRed		 := 254;
		
		byTopRightShelfRed			 := 254;
		byMiddle1RightShelfRed		 := 254;	 
		byMiddle2RightShelfRed		 := 254;	
		byBottomRightShelfRed		 := 254;
	END_IF
	
	IF FBEnOceanPTM200[2].bSwitches[1] THEN
		byTopLeftShelfGreen				 := 254;
		byMiddle1LeftShelfGreen			 := 254;	 
		byMiddle2LeftShelfGreen			 := 254;	
		byBottomLeftShelfGreen			 := 254;
		
		byTopRightShelfGreen			 := 254;
		byMiddle1RightShelfGreen		 := 254;	 
		byMiddle2RightShelfGreen		 := 254;	
		byBottomRightShelfGreen			 := 254;
	END_IF

	IF FBEnOceanPTM200[2].bSwitches[2] THEN
		byTopLeftShelfBlue				 := 254;
		byMiddle1LeftShelfBlue			 := 254;	 
		byMiddle2LeftShelfBlue			 := 254;	
		byBottomLeftShelfBlue			 := 254;
		
		byTopRightShelfBlue				 := 254;
		byMiddle1RightShelfBlue			 := 254;	 
		byMiddle2RightShelfBlue			 := 254;	
		byBottomRightShelfBlue			 := 254;
	END_IF
	
	IF FBEnOceanPTM200[2].bSwitches[3] OR PTM200StrippedTables[5].Signal THEN
		byTopLeftShelfRed				 := 0;
		byMiddle1LeftShelfRed			 := 0;	 
		byMiddle2LeftShelfRed			 := 0;	
		byBottomLeftShelfRed			 := 0;
		
		byTopRightShelfRed				 := 0;
		byMiddle1RightShelfRed			 := 0;	 
		byMiddle2RightShelfRed			 := 0;	
		byBottomRightShelfRed			 := 0;
		
		byTopLeftShelfGreen				 := 0;
		byMiddle1LeftShelfGreen			 := 0;	 
		byMiddle2LeftShelfGreen			 := 0;	
		byBottomLeftShelfGreen			 := 0;
		
		byTopRightShelfGreen			 := 0;
		byMiddle1RightShelfGreen		 := 0;	 
		byMiddle2RightShelfGreen		 := 0;	
		byBottomRightShelfGreen			 := 0;
		
		byTopLeftShelfBlue				 := 0;
		byMiddle1LeftShelfBlue			 := 0;	 
		byMiddle2LeftShelfBlue			 := 0;	
		byBottomLeftShelfBlue			 := 0;
		
		byTopRightShelfBlue				 := 0;
		byMiddle1RightShelfBlue			 := 0;	 
		byMiddle2RightShelfBlue			 := 0;	
		byBottomRightShelfBlue			 := 0;
	END_IF

	// SET DMX Shelves for Projector Mode
	IF FBEnOceanPTM200[0].bSwitches[2] THEN
		byTopLeftShelfRed				 := 0;
		byMiddle1LeftShelfRed			 := 0;	 
		byMiddle2LeftShelfRed			 := 0;	
		byBottomLeftShelfRed			 := 0;
		byTopRightShelfRed				 := 0;
		byMiddle1RightShelfRed			 := 0;	 
		byMiddle2RightShelfRed			 := 0;	
		byBottomRightShelfRed			 := 0;
		
		byTopLeftShelfGreen				 := 0;
		byMiddle1LeftShelfGreen			 := 0;	 
		byMiddle2LeftShelfGreen			 := 0;	
		byBottomLeftShelfGreen			 := 0;
		byTopRightShelfGreen			 := 0;
		byMiddle1RightShelfGreen		 := 0;	 
		byMiddle2RightShelfGreen		 := 0;	
		byBottomRightShelfGreen			 := 0;
		
		byTopLeftShelfBlue				 := 254;
		byMiddle1LeftShelfBlue			 := 254;	 
		byMiddle2LeftShelfBlue			 := 254;	
		byBottomLeftShelfBlue			 := 254;
		byTopRightShelfBlue				 := 254;
		byMiddle1RightShelfBlue			 := 254;	 
		byMiddle2RightShelfBlue			 := 254;	
		byBottomRightShelfBlue			 := 254;
	END_IF
	
hmiUpdateTimer(enable:= TRUE, offTime:= T#0.5S, onTime:= T#0.5S, Q=> updateHmi);	

//Selected shelves get RGB value from HMI colour picker	
(*LEFT SIDE OF CABINET*)
IF shelfSelection[1] THEN
	byTopLeftShelfRed			:= colours.red;
	byTopLeftShelfGreen			:= colours.green;
	byTopLeftShelfBlue			:= colours.blue;
END_IF                      	
                            	
IF shelfSelection[2] THEN   	
	byMiddle1LeftShelfRed		:= colours.red;
	byMiddle1LeftShelfGreen		:= colours.green;
	byMiddle1LeftShelfBlue		:= colours.blue;
END_IF                      	
                            	
IF shelfSelection[3] THEN   	
	byMiddle2LeftShelfRed		:= colours.red;
	byMiddle2LeftShelfGreen		:= colours.green;
	byMiddle2LeftShelfBlue		:= colours.blue;
END_IF                      	
                            	
IF shelfSelection[4] THEN   	
	byBottomLeftShelfRed		:= colours.red;
	byBottomLeftShelfGreen		:= colours.green;
	byBottomLeftShelfBlue		:= colours.blue;
END_IF                      	
                            	
(*RIGHT SIDE OF CABINET*)   	
IF shelfSelection[5] THEN   	
	byTopRightShelfRed			:= colours.red;
	byTopRightShelfGreen		:= colours.green;
	byTopRightShelfBlue			:= colours.blue;
END_IF                      	
                            	
IF shelfSelection[6] THEN   	
	byMiddle1RightShelfRed		:= colours.red;
	byMiddle1RightShelfGreen	:= colours.green;
	byMiddle1RightShelfBlue		:= colours.blue;
END_IF                      	
                            	
IF shelfSelection[7] THEN   	
	byMiddle2RightShelfRed		:= colours.red;
	byMiddle2RightShelfGreen	:= colours.green;
	byMiddle2RightShelfBlue		:= colours.blue;
END_IF                      	
                            	
IF shelfSelection[8] THEN   	
	byBottomRightShelfRed		:= colours.red;
	byBottomRightShelfGreen		:= colours.green;
	byBottomRightShelfBlue		:= colours.blue;
END_IF

ACTION MoveDMXValues:

	//Left Shelf					
	arrDMXProcessData[1] := byTopLeftShelfRed;
	arrDMXProcessData[2] := byTopLeftShelfGreen;
	arrDMXProcessData[3] := byTopLeftShelfBlue;

	arrDMXProcessData[10] := byMiddle1LeftShelfRed;
	arrDMXProcessData[11] := byMiddle1LeftShelfGreen;
	arrDMXProcessData[12] := byMiddle1LeftShelfBlue;

	arrDMXProcessData[20] := byMiddle2LeftShelfRed;
	arrDMXProcessData[21] := byMiddle2LeftShelfGreen;
	arrDMXProcessData[22] := byMiddle2LeftShelfBlue;

	arrDMXProcessData[30] := byBottomLeftShelfRed;
	arrDMXProcessData[31] := byBottomLeftShelfGreen;
	arrDMXProcessData[32] := byBottomLeftShelfBlue;

	
	//Right Shelf
	arrDMXProcessData[40] := byTopRightShelfRed;
	arrDMXProcessData[41] := byTopRightShelfGreen;
	arrDMXProcessData[42] := byTopRightShelfBlue;

	arrDMXProcessData[50] := byMiddle1RightShelfRed;
	arrDMXProcessData[51] := byMiddle1RightShelfGreen;
	arrDMXProcessData[52] := byMiddle1RightShelfBlue;

	arrDMXProcessData[60] := byMiddle2RightShelfRed;
	arrDMXProcessData[61] := byMiddle2RightShelfGreen;
	arrDMXProcessData[62] := byMiddle2RightShelfBlue;

	arrDMXProcessData[70] := byBottomRightShelfRed;
	arrDMXProcessData[71] := byBottomRightShelfGreen;
	arrDMXProcessData[72] := byBottomRightShelfBlue;
END_ACTION

END_PROGRAM

// ---- WORKSHOP WALL/Pulse.TcPOU
FUNCTION_BLOCK Pulse
VAR_INPUT
	enable		:	BOOL;
	offTime		:	TIME;
	onTime		:	TIME;
END_VAR
VAR_OUTPUT
	Q			:	BOOL;
END_VAR
VAR
	onTimer		:	TON;
	offTimer	:	TON;
END_VAR

offTimer(IN:= enable AND NOT(onTimer.Q), PT:= offTime, Q=> Q, ET=> );

onTimer(IN:= offTimer.Q, PT:= onTime, Q=> , ET=> );

END_FUNCTION_BLOCK

// ---- MAIN.TcPOU
PROGRAM MAIN
VAR
	
	BasicTestingEnabled					: BOOL;
                            			
	FB_BlindControl						: ARRAY [0..2] OF BlindControl;
                            			
	i									: INT;
                            			
	bTest								: BOOL;
	bLog								: BOOL;
                    					
	arrData								: ARRAY[0..BUFFER_SIZE] OF ST_PHASE_DATA;
	arrSnapshotData						: ARRAY[0..BUFFER_SIZE] OF ST_PHASE_DATA;
                    					
	iState								: INT;
	bExecute							: BOOL;
	bBusy								: BOOL;
                            	
	bError 								: BOOL;
	tonSampleRate						: TON;

	aDataPacket1						: ARRAY [0..6] OF BYTE := [16#9A, 16#04, 16#00, 16#00, 16#0A, 16#00, 16#00]; 		(* Main office *)
	aDataPacket2						: ARRAY [0..6] OF BYTE :=  [16#9A, 16#02, 16#00, 16#00, 16#0A, 16#00, 16#00];		(* Board Room*)
	aDataPacket3						: ARRAY [0..6] OF BYTE := [16#9A, 16#03, 16#00, 16#00, 16#0A, 16#00, 16#00]; 		(* Reception *)
	
	
	bStretch							: BOOL;
	bStretchDone						: BOOL;
	HowOftenTimer						: Ton := (PT:= T#21d);//31d);
		
	fbBlindsStretch						: BlindStretch;

	hmiStrech							: BOOL;
	
	fbWindSimulator						: FB_WindTurbineSim;
	
	windSpeed							: LREAL;
	
	bGetOpenWeatherMap             		: BOOL;

    fbHttpClientOpenWeatherMap     		: FB_IotHttpClient :=(sHostName:='api.weatherapi.com', bKeepAlive:=TRUE, tConnectionTimeout:=T#10S);

    fbWeatherAPI        				: FB_WeatherAPI_HTTP;
	
	fbSendWatsappCallMeBot				: FB_SendWhatsappCallMeBot;
	
	fbHttpClientWhatsAppResponse   		: FB_IotHttpClient :=(sHostName:='webhook.site', bKeepAlive:=TRUE, tConnectionTimeout:=T#10S);
	
	fbWhatsAppRespose					: FB_WatsAppResponse;
	
	textWhatsApp						: T_MaxString;
	
	weatherTon							: ton := (pt:=T#10m);					
	local: BOOL;
	hmiFinished: BOOL;
	testWhatsApp: BOOL;
END_VAR

BackgroundComms();
ADSReadCX9020();
EnOcean();
//SQLDB();
PrgMqttCom_PM_Subscriber();
//PrgMqttCom_Blinds_Publisher();
//CoffeePredictionML();
//MLtest();
Dali();
//DMX();
LightControl();
//ReadCP67();
FileHandle();
TableTennisScoreCounter();
VariableHandleForHmi();
SleepModeCheck();
PowerSupply();

FB_BlindControl[0](
	BulkCommand:= BackgroundComms.BlindCommandTable[0].SelectBlindsBulkCommand ,
	xCommandUp:= BackgroundComms.BlindCommandTable[0].xCommandUp,
	xCommandDown:= BackgroundComms.BlindCommandTable[0].xCommandDown ,
	xCommandStop:= BackgroundComms.BlindCommandTable[0].xCommandStop ,
	HubTXBuffer:= BackgroundComms.HubTXBuffer[0] ,
	HubRXBuffer:= BackgroundComms.HubRXBuffer[0] ,
	aDataPacket := aDataPacket1,
	xCommandUpJog := BackgroundComms.BlindCommandTable[0].xCommandUpJog ,
	xCommandDownJog := BackgroundComms.BlindCommandTable[0].xCommandDownJog ,
	JogTime :=  BackgroundComms.BlindCommandTable[0].JogTime,
	JogTimeInt :=  BackgroundComms.BlindCommandTable[0].JogTimeInt,
	xBusy => );

FB_BlindControl[1](
	BulkCommand:= BackgroundComms.BlindCommandTable[1].SelectBlindsBulkCommand ,
	xCommandUp:= BackgroundComms.BlindCommandTable[1].xCommandUp,
	xCommandDown:= BackgroundComms.BlindCommandTable[1].xCommandDown ,
	xCommandStop:= BackgroundComms.BlindCommandTable[1].xCommandStop ,
	HubTXBuffer:= BackgroundComms.HubTXBuffer[1] ,
	HubRXBuffer:= BackgroundComms.HubRXBuffer[1] ,
	aDataPacket :=  aDataPacket2,
	xCommandUpJog := BackgroundComms.BlindCommandTable[1].xCommandUpJog ,
	xCommandDownJog := BackgroundComms.BlindCommandTable[1].xCommandDownJog ,
	JogTime :=  BackgroundComms.BlindCommandTable[1].JogTime,
	JogTimeInt :=  BackgroundComms.BlindCommandTable[1].JogTimeInt,
	xBusy => );

FB_BlindControl[2](
	BulkCommand:= BackgroundComms.BlindCommandTable[2].SelectBlindsBulkCommand ,
	xCommandUp:= BackgroundComms.BlindCommandTable[2].xCommandUp,
	xCommandDown:= BackgroundComms.BlindCommandTable[2].xCommandDown ,
	xCommandStop:= BackgroundComms.BlindCommandTable[2].xCommandStop ,
	HubTXBuffer:= BackgroundComms.HubTXBuffer[2] ,
	HubRXBuffer:= BackgroundComms.HubRXBuffer[2] ,
	aDataPacket :=  aDataPacket3,
	xCommandUpJog := BackgroundComms.BlindCommandTable[2].xCommandUpJog ,
	xCommandDownJog := BackgroundComms.BlindCommandTable[2].xCommandDownJog ,
	JogTime :=  BackgroundComms.BlindCommandTable[2].JogTime,
	JogTimeInt :=  BackgroundComms.BlindCommandTable[2].JogTimeInt,
	xBusy => );
	

HowOftenTimer.IN:= TRUE;

IF HowOftenTimer.Q THEN
	bStretch := TRUE;
	hmiFinished := FALSE;
END_IF

IF bStretchDone THEN
	HowOftenTimer.IN := FALSE;
	bStretchDone := FALSE;
	bStretch := FALSE;
	hmiStrech := FALSE;
	hmiFinished := TRUE;
END_IF
	
fbBlindsStretch(Start:= bStretch AND hmiStrech, StretchDone:= bStretchDone,Err=> );

HowOftenTimer();

IF NOT fbHttpClientOpenWeatherMap.bConfigured THEN
    fbHttpClientOpenWeatherMap.nHostPort:= 443;
    fbHttpClientOpenWeatherMap.stTLS.bNoServerCertCheck:= TRUE;
	weatherTon.IN := TRUE;
END_IF

IF fbHttpClientOpenWeatherMap.bConfigured THEN
    fbWeatherAPI(bSend:=weatherTon.Q, fbClient:=fbHttpClientOpenWeatherMap);
END_IF

IF weatherTon.Q THEN
	weatherTon.IN := FALSE;
ELSE
	weatherTon.IN := TRUE;
END_IF

fbHttpClientOpenWeatherMap.Execute();
WindSpeed := fbWeatherAPI.wind_speed;
fbWindSimulator(windSpeed:= WindSpeed, rpm=> RPM, powerOutput=> Power);
weatherTon();

fbSendWatsappCallMeBot(SendText := , YourNumber := '447724278323', Text2Send := textWhatsApp, ApiKey := '6082625');  //SendText := , YourNumber := '+447724278323', Text2Send := textWhatsApp, ApiKey := 'US6Y79pt7LAU'

IF testWhatsApp THEN	//RPM > 200 AND weatherTon.Q 
	textWhatsApp := 'Wind turbine at risk, consider switching the turbine off.';
	fbSendWatsappCallMeBot.SendText := TRUE;
ELSE
	fbSendWatsappCallMeBot.SendText := FALSE;
END_IF

IF NOT fbHttpClientWhatsAppResponse.bConfigured THEN
    fbHttpClientOpenWeatherMap.nHostPort:= 443;
    fbHttpClientOpenWeatherMap.stTLS.bNoServerCertCheck:= TRUE;
	//weatherTon.IN := TRUE;
END_IF

IF fbHttpClientWhatsAppResponse.bConfigured THEN
    fbWhatsAppRespose(bSend:=testWhatsApp, fbClient:=fbHttpClientWhatsAppResponse);
END_IF

fbHttpClientWhatsAppResponse.Execute();

ACTION SleepModeCheck:
IF Global_Variables.xSleepMode THEN
	
	// Set Socket State
	xXplanarScreenPowerOff := TRUE;
	
		

	xSleepMode := FALSE;						// Reset Sleep Call	
	
END_IF
END_ACTION

END_PROGRAM

// ---- BLINDS/BlindStretch.TcPOU
FUNCTION_BLOCK BlindStretch
VAR_INPUT
	Start						: BOOL;
END_VAR                 		  
VAR_OUTPUT              		  
	Err							: BOOL;
END_VAR                 		  
VAR                         	
	UpdateInterval				: BYTE;      	  
	fbBlindsControl				: BlindControl;
	GetBusyBitOffice			: ADSREADEX := ( NETID := '5.129.86.232.1.1', PORT := 851, TMOUT := T#5S );
	GetBusyBitKitchen			: ADSREADEX := ( NETID := '5.129.86.232.1.1', PORT := 851, TMOUT := T#5S );
	GetBusyBitBoardroom			: ADSREADEX := ( NETID := '5.129.86.232.1.1', PORT := 851, TMOUT := T#5S );
	                    		  
	BusyOffice					: BOOL;
	BusyKitchen					: BOOL;
	BusyBoardroom				: BOOL;
	                        	
	testInt						: int;
	                        	
	BusyBits					: ARRAY[0..2] OF BOOL;
	
	
	
	//BlindSelector			: INT;
	
	//BlindSelector		AT%M*	: INT;
	                    		  
	TonError					: Ton := (PT := T#30S);
	TonUpCommand				: Ton;
	TonDownCommand				: Ton;
	                        	
	iState						: INT;
END_VAR                     	
                            	
VAR_IN_OUT                  	
	StretchDone					: BOOL;
END_VAR

UpdateInterval := UpdateInterval + 1;

		GetBusyBitOffice(
			NETID:= '5.129.86.232.1.1',
			PORT:= 851 ,
			IDXGRP:=16#4040,//16#4020 ,
			IDXOFFS:= 16#6DD89,//0,
			LEN:= 4,//40,
			DESTADDR:= ADR(BusyBits[0]),
			READ:= UpdateInterval.0,
			TMOUT:= t#5s,
			BUSY=> ,
			ERR=> ,
			ERRID=> ,
			COUNT_R=> );
			
		GetBusyBitBoardroom(
			NETID:= '5.129.86.232.1.1',
			PORT:= 851 ,
			IDXGRP:=16#4040,//16#4020 ,
			IDXOFFS:= 16#6DDA9,//0,
			LEN:= 4,//40,
			DESTADDR:= ADR(BusyBits[1]),
			READ:= UpdateInterval.0,
			TMOUT:= t#5s,
			BUSY=> ,
			ERR=> ,
			ERRID=> ,
			COUNT_R=> );
			
		GetBusyBitKitchen(
			NETID:= '5.129.86.232.1.1',
			PORT:= 851 ,
			IDXGRP:=16#4040,//16#4020 ,
			IDXOFFS:= 16#6DDC9,//0,
			LEN:= 4,//40,
			DESTADDR:= ADR(BusyBits[2]),
			READ:= UpdateInterval.0,
			TMOUT:= t#5s,
			BUSY=> ,
			ERR=> ,
			ERRID=> ,
			COUNT_R=> );		

IF Start THEN

CASE iState OF
	0: //Check Busy state if busy for 30+s 100 err or 10

		BlindSelector := 0;
		//BlinderSelection := 0;
		iState := 10;

	10://Select room to be stretched 11 -> offce 12 -> kitchen 13 -> board room
		IF (NOT BusyBits[0] AND NOT BusyBits[1] AND NOT BusyBits[2]) THEN
			//state 10
			TonError.IN := FALSE;
			iState := 11;
			
		ELSE
			//timer for 30 sec -> state 100
			TonError.IN := TRUE;
			IF TonError.Q THEN
				iState := 100;
			END_IF
			
		END_IF
	11://Select individual blinds -> 20 stretch up -> 21 check -> 30 strech down -> 31 check -> 40 stretch up -> 41 check
		BlindCX7000UserTable[BlindSelector].SelectBlindsBulkCommand[1] := TRUE;
		BlindCX7000UserTable[BlindSelector].SelectBlindsBulkCommand[2] := TRUE; 
		BlindCX7000UserTable[BlindSelector].SelectBlindsBulkCommand[3] := TRUE; 
		BlindCX7000UserTable[BlindSelector].SelectBlindsBulkCommand[4] := TRUE; 
		BlindCX7000UserTable[BlindSelector].SelectBlindsBulkCommand[5] := TRUE; 
		BlindCX7000UserTable[BlindSelector].SelectBlindsBulkCommand[6] := TRUE; 
		BlindCX7000UserTable[BlindSelector].SelectBlindsBulkCommand[7] := TRUE; 
		BlindCX7000UserTable[BlindSelector].SelectBlindsBulkCommand[8] := TRUE; 
		BlindCX7000UserTable[BlindSelector].SelectBlindsBulkCommand[9] := TRUE; 
		BlindCX7000UserTable[BlindSelector].SelectBlindsBulkCommand[10] := TRUE;
		BlindCX7000UserTable[BlindSelector].SelectBlindsBulkCommand[11] := True;
		BlindCX7000UserTable[BlindSelector].SelectBlindsBulkCommand[12] := True;
		BlindCX7000UserTable[BlindSelector].SelectBlindsBulkCommand[13] := True;
		BlindCX7000UserTable[BlindSelector].SelectBlindsBulkCommand[14] := True;
		BlindCX7000UserTable[BlindSelector].SelectBlindsBulkCommand[15] := True;
		BlindCX7000UserTable[BlindSelector].SelectBlindsBulkCommand[16] := True;
		
		iState := 20;
		
	12://Select individual blinds -> 20 stretch up -> 21 check -> 30 strech down -> 31 check -> 40 stretch up -> 41 check
		BlindCX7000UserTable[BlindSelector].SelectBlindsBulkCommand[1] := TRUE;
		BlindCX7000UserTable[BlindSelector].SelectBlindsBulkCommand[2] := TRUE; 
		BlindCX7000UserTable[BlindSelector].SelectBlindsBulkCommand[3] := TRUE; 
		BlindCX7000UserTable[BlindSelector].SelectBlindsBulkCommand[4] := TRUE; 
		BlindCX7000UserTable[BlindSelector].SelectBlindsBulkCommand[5] := TRUE; 
		BlindCX7000UserTable[BlindSelector].SelectBlindsBulkCommand[6] := TRUE; 
		BlindCX7000UserTable[BlindSelector].SelectBlindsBulkCommand[7] := TRUE; 
		BlindCX7000UserTable[BlindSelector].SelectBlindsBulkCommand[8] := True; 
		BlindCX7000UserTable[BlindSelector].SelectBlindsBulkCommand[9] := True; 
		BlindCX7000UserTable[BlindSelector].SelectBlindsBulkCommand[10] := TRUE;
		BlindCX7000UserTable[BlindSelector].SelectBlindsBulkCommand[11] := TRUE;
		BlindCX7000UserTable[BlindSelector].SelectBlindsBulkCommand[12] := TRUE;
		BlindCX7000UserTable[BlindSelector].SelectBlindsBulkCommand[13] := TRUE;
		BlindCX7000UserTable[BlindSelector].SelectBlindsBulkCommand[14] := TRUE;
		BlindCX7000UserTable[BlindSelector].SelectBlindsBulkCommand[15] := TRUE;
		BlindCX7000UserTable[BlindSelector].SelectBlindsBulkCommand[16] := TRUE;
		
		iState := 20;
		
	13://Select individual blinds -> 20 stretch up -> 21 check -> 30 strech down -> 31 check -> 40 stretch up -> 41 check
		BlindCX7000UserTable[BlindSelector].SelectBlindsBulkCommand[1] := TRUE;
		BlindCX7000UserTable[BlindSelector].SelectBlindsBulkCommand[2] := TRUE; 
		BlindCX7000UserTable[BlindSelector].SelectBlindsBulkCommand[3] := TRUE; 
		BlindCX7000UserTable[BlindSelector].SelectBlindsBulkCommand[4] := TRUE; 
		BlindCX7000UserTable[BlindSelector].SelectBlindsBulkCommand[5] := TRUE; 
		BlindCX7000UserTable[BlindSelector].SelectBlindsBulkCommand[6] := TRUE; 
		BlindCX7000UserTable[BlindSelector].SelectBlindsBulkCommand[7] := TRUE; 
		BlindCX7000UserTable[BlindSelector].SelectBlindsBulkCommand[8] := TRUE; 
		BlindCX7000UserTable[BlindSelector].SelectBlindsBulkCommand[9] := TRUE; 
		BlindCX7000UserTable[BlindSelector].SelectBlindsBulkCommand[10] := TRUE;
		BlindCX7000UserTable[BlindSelector].SelectBlindsBulkCommand[11] := TRUE;
		BlindCX7000UserTable[BlindSelector].SelectBlindsBulkCommand[12] := TRUE;
		BlindCX7000UserTable[BlindSelector].SelectBlindsBulkCommand[13] := TRUE;
		BlindCX7000UserTable[BlindSelector].SelectBlindsBulkCommand[14] := TRUE;
		BlindCX7000UserTable[BlindSelector].SelectBlindsBulkCommand[15] := TRUE;
		BlindCX7000UserTable[BlindSelector].SelectBlindsBulkCommand[16] := TRUE;
		
		iState := 20;
	20://Strech up for X seconds
		TonUpCommand.IN := TRUE;
		TonUpCommand.PT := T#30S;

		IF NOT BusyBits[BlindSelector] THEN
			BlindCX7000UserTable[BlindSelector].xCommandUp := TRUE;
		ELSE
			BlindCX7000UserTable[BlindSelector].xCommandUp := FALSE;
			iState := 201;
		END_IF
		
	201:
		IF TonUpCommand.Q THEN
			IF NOT BusyBits[BlindSelector] THEN
				BlindCX7000UserTable[BlindSelector].xCommandStop := TRUE;
			ELSE
				BlindCX7000UserTable[BlindSelector].xCommandStop := FALSE;
				TonUpCommand.IN := FALSE;
				iState := 21;
			END_IF
		END_IF
		
	202:
		IF NOT BusyBits[BlindSelector] THEN
			BlindCX7000UserTable[BlindSelector].xCommandStop := TRUE;
		ELSE
			BlindCX7000UserTable[BlindSelector].xCommandStop := FALSE;
			iState := 8;
		END_IF

	21://Check if busy
		IF BlindSelector = 0 THEN
			IF NOT BusyBits[BlindSelector] THEN
				iState := 30;
			END_IF
		ELSIF BlindSelector = 1 THEN
			IF NOT BusyBits[BlindSelector] THEN
				iState := 30;
			END_IF
		ELSIF BlindSelector = 2 THEN
			IF NOT BusyBits[BlindSelector] THEN
				iState := 30;
			END_IF
		END_IF 
	30://Strech down for Y seconds
		TonDownCommand.IN := TRUE;
		TonDownCommand.PT := T#30S;
		
		IF NOT BusyBits[BlindSelector] THEN
			BlindCX7000UserTable[BlindSelector].xCommandDown := TRUE;
		ELSE
			BlindCX7000UserTable[BlindSelector].xCommandDown := FALSE;
			iState := 301;
		END_IF	
		
	301:
		IF TonDownCommand.Q THEN
			IF NOT BusyBits[BlindSelector] THEN
				BlindCX7000UserTable[BlindSelector].xCommandStop := TRUE;
			ELSE
				BlindCX7000UserTable[BlindSelector].xCommandStop := FALSE;
				TonDownCommand.IN := FALSE;
				iState := 31;
			END_IF
		END_IF
	
		
//		nState := 31;
	31://Check if Busy
		IF BlindSelector = 0 THEN
			IF NOT BusyBits[BlindSelector] THEN
				iState := 40;
			END_IF
		ELSIF BlindSelector = 1 THEN
			IF NOT BusyBits[BlindSelector] THEN
				iState := 40;
			END_IF
		ELSIF BlindSelector = 2 THEN
			IF NOT BusyBits[BlindSelector] THEN
				iState := 40;
			END_IF
		END_IF 
	40://Strech up for X seconds
		TonUpCommand.IN := TRUE;
		TonUpCommand.PT := T#30S;
		IF NOT BusyBits[BlindSelector] THEN
			BlindCX7000UserTable[BlindSelector].xCommandUp := TRUE;
		ELSE
			BlindCX7000UserTable[BlindSelector].xCommandUp := FALSE;
			iState := 401;
		END_IF
	
	401:
		IF TonUpCommand.Q THEN
			IF NOT BusyBits[BlindSelector] THEN
				BlindCX7000UserTable[BlindSelector].xCommandStop := TRUE;
			ELSE
				BlindCX7000UserTable[BlindSelector].xCommandStop := FALSE;
				TonUpCommand.IN := FALSE;
				iState := 41;
			END_IF
		END_IF	
		
	41://Check if busy
		IF BlindSelector = 0 THEN
			IF NOT BusyBits[BlindSelector] THEN
				BlindSelector := 1;
				iState := 12;
			END_IF
		ELSIF BlindSelector = 1 THEN
			IF NOT BusyBits[BlindSelector] THEN
				BlindSelector := 2;
				iState := 13;
			END_IF
		ELSIF BlindSelector = 2 THEN
			IF NOT BusyBits[BlindSelector] THEN
				StretchDone := TRUE;
				iState := 0;
			END_IF
		END_IF 
	100://Err handling
	
END_CASE
	
//time out strech up

//time out strech down

//time out stretch up
	
END_IF
//HowOftenTimer();
TonError();
TonUpCommand();
TonDownCommand();

END_FUNCTION_BLOCK

// ---- WIND TURBINE/FB_WindTurbineSim.TcPOU
FUNCTION_BLOCK FB_WindTurbineSim
VAR_INPUT
	windSpeed		: LREAL;
	
END_VAR
VAR_OUTPUT
	rpm				: LREAL;
	powerOutput		: LREAL;
END_VAR
VAR
	risingCoef		: LREAL := 0.000314; //Coefficient for the rising segment for SD6+
	tipSpeed		: LREAL;
	cutInSpeed		: LREAL := 5.59234;	//mph
	
END_VAR

VAR CONSTANT
	radius			: LREAL := 2.8;		//5.6m diameter of SD Wind SD6+ turbine
	tsr				: Lreal	:= 2.5;		//tip speed ration usually arownd 7 for commercial turbines
	maxRPM			: LREAL	:= 200.0;
	maxOperationalSpeed: LREAL := 156.586;	//mph
	ratedSpeed		: LREAL := 30;			//mph
END_VAR

IF windSpeed < 6.00 THEN
	powerOutput := 0.00;
ELSIF windSpeed <= 30.00 THEN
	powerOutput := risingCoef * EXPT(windSpeed, 3);
ELSIF windSpeed <= 55.00 THEN
	powerOutput := 8.5;
ELSE
	powerOutput := 0;
END_IF

IF windSpeed < cutInSpeed THEN
	rpm := 0;
END_IF

IF windSpeed <= ratedSpeed THEN
	tipSpeed := tsr * windSpeed;
	rpm := (tipSpeed * 60) / (3.14 * 2 * radius);
	rpm := MIN(rpm, maxRPM);

ELSE
	rpm := maxRPM;
END_IF

//tipSpeed := tsr * MIN(windSpeed,maxOperationalSpeed);



//IF rpm > maxRPM THEN
//	rpm := maxRPM;
//END_IF

END_FUNCTION_BLOCK

// ---- WIND TURBINE/FB_WeatherAPI_HTTP.TcPOU
FUNCTION_BLOCK FB_WeatherAPI_HTTP
VAR_INPUT
	bSend             : BOOL;
END_VAR
VAR_OUTPUT
	wind_speed		  : Lreal;
	bBusy             : BOOL;
    bError            : BOOL;
END_VAR
VAR
	fbRequest         : FB_IotHttpRequest;
    fbJson            : FB_JsonDomParser;
    nState            : UDINT;
    RisingEdge        : R_TRIG;

    bGetContentResult : BOOL;
    sContent          : STRING(511);

    bGetJsonResult    : BOOL;
    jsonDoc           : SJsonValue;
    jsonVal           : SJsonValue;
	jsonWind           : SJsonValue;

    nReqCount         : UDINT;
    nResCount         : UDINT;
    nValidResCount    : UDINT;
    nErrCount         : UDINT;
	bHasMember		  : BOOL;
	bHasMember2		  : BOOL;
END_VAR
VAR_IN_OUT
	 fbClient          : FB_IotHttpClient;
END_VAR

RisingEdge(CLK:= bSend);
CASE nState OF
0:
    IF RisingEdge.Q THEN
        IF fbRequest.SendRequest(sUri:= '/v1/current.json?q=East%20Kilbride&key=8976e01a943e4ee8915133914242706',
                                 fbClient:= fbClient, 
                                 eRequestType:= ETcIotHttpRequestType.HTTP_Get, 0, 0, 0) THEN
            nState:= 1;
            nReqCount:= nReqCount+1;
            bBusy:= TRUE;
            bError:= FALSE;
        END_IF
    END_IF
1:
    IF NOT fbRequest.bBusy THEN
        bError:= TRUE;
        IF NOT fbRequest.bError THEN
            bGetContentResult:= fbRequest.GetContent(pContent:= ADR(sContent), 
                                                     nContentSize:= SIZEOF(sContent), 
                                                     bSetNullTermination:= TRUE);
            IF fbRequest.nStatusCode >= 200 AND fbRequest.nStatusCode < 300 THEN
                bGetJsonResult:= FALSE;
                jsonDoc:= fbRequest.GetJsonDomContent(fbJson);
                IF jsonDoc <> 0 THEN
                    bHasMember := fbJson.HasMember(jsonDoc, 'current');
					IF (bHasMember) THEN
						bHasMember := FALSE;
						jsonVal := fbJson.FindMember(jsonDoc, 'current');
					END_IF
					
					bHasMember2 := fbJson.HasMember(jsonVal, 'wind_mph');
					IF (bHasMember2) THEN
						bHasMember2 := FALSE;
						jsonWind := fbJson.FindMember(jsonVal, 'wind_mph');
						wind_speed := fbJson.GetDouble(jsonWind);
						WindSpeed := fbJson.GetDouble(jsonWind);
					END_IF
					
                    nValidResCount:= nValidResCount+1;
                    bError:= FALSE;
                END_IF
                nResCount:= nResCount+1;
            END_IF
        END_IF
        nState:= 0;
        bBusy:= FALSE;
        IF bError THEN
            nErrCount:= nErrCount+1;
        END_IF
    END_IF
END_CASE

END_FUNCTION_BLOCK

// ---- WIND TURBINE/FB_SendWhatsappCallMeBot.TcPOU
FUNCTION_BLOCK FB_SendWhatsappCallMeBot
VAR_INPUT
	SendText			: BOOL;
	YourNumber			: T_MaxString;
	Text2Send			: T_MaxString;
	ApiKey				: T_MaxString;
END_VAR
VAR_OUTPUT
END_VAR
VAR
    // trigger command execution for OpenWeatherMap samples
	fbHttpClient		: FB_IotHttpClient :=(sHostName:='api.callmebot.com',
							bKeepAlive:=TRUE, tConnectionTimeout:=T#10S);
	
//	fbHttpClient		: FB_IotHttpClient :=(sHostName:='api.textmebot.com',
//							bKeepAlive:=TRUE, tConnectionTimeout:=T#10S);

    fbRequest           : FB_IotHttpRequest;
							
	// https://api.callmebot.com/whatsapp.php?phone=+324xxxxxxxx&text=This+is+a+test&apikey=yyyyyy
	fbFormatString      : FB_FormatString;
	sConMessage			: STRING(255);
	rtrSend				: R_TRIG;
	
	lText2Send			: T_MaxString;
	ifor				: INT;
END_VAR

fbHttpClient.Execute();



rtrSend(CLK := SendText);	
IF rtrSend.Q THEN
	lText2Send := Text2Send;
	
	// Replace spaces in text to '+'
	FOR ifor := 1 TO len(lText2Send) DO
		IF MID(lText2Send,1,ifor) = ' ' THEN
			lText2Send := REPLACE(lText2Send,'+',1,ifor);
		END_IF
	END_FOR

	fbFormatString(
		sFormat := '/whatsapp.php?phone=%s&text=%s&apikey=%s', //'/send.php?recipient=%s&apikey=%s&text=%s'
		arg1    := F_STRING(YourNumber), 
		arg2    := F_STRING(lText2Send), 
		arg3    := F_STRING(ApiKey), 
		bError  => , 
		nErrId  => , 
		sOut    => sConMessage);

	fbRequest.SendRequest(sUri:=sConMessage, fbClient:=fbHttpClient, eRequestType:=ETcIotHttpRequestType.HTTP_POST, 0, 0, 0);
END_IF

END_FUNCTION_BLOCK

